    MoveJ pInicioX62_Pinca1, V_rapide, Z_arret, Tool_Pince1\WObj:=wobj_X62;
    !
    ! E13:interferencia2 com K5
    ! O12:fora de interferencia1 com K5
    EVENT\E13;
    ORDRE\O12;
    !
    MoveJ [[602.06,1695.19,2908.36],[0.0694316,-0.00204347,0.00124342,-0.997584],[0,-1,0,0],[59.9379,9E+09,9E+09,9E+09,9E+09,9E+09]], V_rapide, Z_arret, Tool_Pince1\WObj:=wobj_X62;
    !
    ! E13:interferencia2 com K5
    ! O12:fora de interferencia1 com K5
    EVENT\E13;
    ORDRE\O12;
    !
    MoveJ [[1650.02,1566.65,2799.96],[0.370322,0.000249773,0.000216744,-0.928904],[0,0,1,0],[15,9E+09,9E+09,9E+09,9E+09,9E+09]], V_rapide, Z_moyen, Tool_Pince1\WObj:=wobj_X62;
    MoveJ [[2181.41,1327.16,2032.09],[0.381242,0.000299882,0.000125925,-0.924475],[0,0,1,0],[183.538,9E+09,9E+09,9E+09,9E+09,9E+09]], V_rapide, Z_moyen, Tool_Pince1\WObj:=wobj_X62;
    MoveL [[1800.58,758.31,2024.83],[0.381244,0.000300867,0.000120671,-0.924474],[0,0,0,0],[183.538,9E+09,9E+09,9E+09,9E+09,9E+09]], V_rapide, Z_moyen, Tool_Pince1\WObj:=wobj_X62;
    MoveL [[1764.11,614.16,2072.30],[0.381245,0.000303532,0.00010268,-0.924474],[0,0,0,0],[183.538,9E+09,9E+09,9E+09,9E+09,9E+09]], V_rapide, Z_moyen, Tool_Pince1\WObj:=wobj_X62;
    MoveL [[1659.86,663.46,2032.41],[0.381237,0.000301139,0.000117928,-0.924477],[0,0,0,0],[140,9E+09,9E+09,9E+09,9E+09,9E+09]], V_rapide, Z_moyen, Tool_Pince1\WObj:=wobj_X62;
    !
    SR_SOUDER lscs2002942400,V_moyen,1,1,Tool_Pince1,wobj_X62;
    SR_SOUDER lscsg002940402,V_moyen,1,2,Tool_Pince1,wobj_X62;
    SR_SOUDER lscsg002940502,V_moyen,1,2,Tool_Pince1,wobj_X62;
    !
    MoveL [[1888.73,628.89,2158.57],[0.46006,-0.0228879,-0.0118518,-0.887514],[0,-1,0,0],[35.0008,9E+09,9E+09,9E+09,9E+09,9E+09]],V_rapide,Z_moyen,Tool_Pince1\WObj:=wobj_X62;
    MoveL [[2001.09,630.15,2158.77],[0.45992,-0.0313939,-0.0162592,-0.887256],[0,-1,0,0],[35,9E+09,9E+09,9E+09,9E+09,9E+09]],V_rapide,Z_moyen,Tool_Pince1\WObj:=wobj_X62;
    !
    SR_SOUDER lscsg002940602,V_moyen,1,2,Tool_Pince1,wobj_X62;
    SR_SOUDER lscsg002940702,V_moyen,1,2,Tool_Pince1,wobj_X62;
    SR_SOUDER lsdcd002932302, V_moyen, 1, 2, Tool_Pince1, wobj_X62;
    !
    MoveL [[2112.35,622.94,2071.75],[0.601153,0.000260756,1.84552E-05,-0.799134],[0,0,0,0],[134.461,9E+09,9E+09,9E+09,9E+09,9E+09]],V_rapide,Z_moyen,Tool_Pince1\WObj:=wobj_X62;
    MoveL [[2277.78,623.66,2088.68],[0.61438,0.00026062,0.000197661,-0.789011],[0,0,0,0],[99.9998,9E+09,9E+09,9E+09,9E+09,9E+09]],V_rapide,Z_moyen,Tool_Pince1\WObj:=wobj_X62;
    !
    SR_SOUDER lscsg002940802_B,V_moyen,1,2,Tool_Pince1,wobj_X62;
    SR_SOUDER lscsg002940902,V_moyen,1,2,Tool_Pince1,wobj_X62;
    SR_SOUDER lscsg002941002,V_moyen,1,2,Tool_Pince1,wobj_X62;
    !
    MoveL [[2430.75,632.00,2159.24],[0.65197,-0.0151493,-0.013018,-0.757982],[0,-1,0,0],[35,9E+09,9E+09,9E+09,9E+09,9E+09]],V_rapide,Z_moyen,Tool_Pince1\WObj:=wobj_X62;
    MoveL [[2543.78,631.39,2158.47],[0.712277,-0.0103391,-0.0104878,-0.701745],[0,-1,0,0],[34.9994,9E+09,9E+09,9E+09,9E+09,9E+09]],V_rapide,Z_moyen,Tool_Pince1\WObj:=wobj_X62;
    !
    SR_SOUDER lscsg002941202,V_moyen,1,2,Tool_Pince1,wobj_X62;
    !
    MoveL [[2540.85,667.11,2064.42],[0.712277,-0.0103403,-0.0104873,-0.701745],[0,-1,0,0],[168.705,9E+09,9E+09,9E+09,9E+09,9E+09]],V_rapide,Z_moyen,Tool_Pince1\WObj:=wobj_X62;
    MoveL [[2529.75,106.99,2062.78],[0.770678,0.00010718,-5.65434E-05,-0.637225],[0,-1,0,0],[170,9E+09,9E+09,9E+09,9E+09,9E+09]],V_rapide,Z_moyen,Tool_Pince1\WObj:=wobj_X62;
    MoveL [[2798.87,290.44,2173.09],[0.872979,-0.00143955,-0.00186681,-0.487753],[0,-1,-1,0],[44.59,9E+09,9E+09,9E+09,9E+09,9E+09]],V_rapide,Z_arret,Tool_Pince1\WObj:=wobj_X62;
    !
    ! O12:fora de interferencia1 com K5
    ! O13:fora de interferencia2 com K5
    ORDRE\O12\O13;
    !
    MoveL [[2687.98,421.61,2066.53],[0.897783,-0.00356194,-0.00758891,-0.440358],[0,0,-1,0],[170,9E+09,9E+09,9E+09,9E+09,9E+09]],V_rapide,Z_moyen,Tool_Pince1\WObj:=wobj_X62;
    MoveL [[2646.63,666.42,2060.91],[0.921929,-0.00569541,-0.013042,-0.387097],[0,0,-1,0],[160,9E+09,9E+09,9E+09,9E+09,9E+09]],V_rapide,Z_moyen,Tool_Pince1\WObj:=wobj_X62;
    !
    SR_SOUDER lscsg002941302,V_moyen,1,2,Tool_Pince1,wobj_X62;
    !
    MoveL [[2646.63,666.42,2060.91],[0.921929,-0.00569541,-0.013042,-0.387097],[0,0,-1,0],[160,9E+09,9E+09,9E+09,9E+09,9E+09]],V_rapide,Z_moyen,Tool_Pince1\WObj:=wobj_X62;
    MoveL [[2638.67,603.72,2062.9],[0.91586,-9.21472E-05,0.000138523,-0.401498],[0,-1,-1,0],[160,9E+09,9E+09,9E+09,9E+09,9E+09]],V_rapide,Z_moyen,Tool_Pince1\WObj:=wobj_X62;
    MoveL [[2733.77,618.85,2085.50],[0.930262,-0.000109742,0.000151233,-0.366895],[0,-1,-1,0],[160,9E+09,9E+09,9E+09,9E+09,9E+09]], V_rapide, Z_arret, Tool_Pince1\WObj:=wobj_X62;
    !
    ! E12:interferencia1 com K5
    ! O13:fora de interferencia2 com K5
    EVENT\E12;
    ORDRE\O13;
    !
    SR_SOUDER lscs2002948300,V_moyen,1,1,Tool_Pince1,wobj_X62;
    SR_SOUDER lscs2002947600, V_moyen, 1, 1, Tool_Pince1, wobj_X62;
    SR_SOUDER lscs2002948400,V_moyen,1,1,Tool_Pince1,wobj_X62;
    !
    MoveL [[2836.77,664.37,2084.41],[0.930318,-0.000108518,0.000131406,-0.366754],[0,-1,-1,0],[100,9E+09,9E+09,9E+09,9E+09,9E+09]],V_rapide,Z_moyen,Tool_Pince1\WObj:=wobj_X62;
    MoveL [[2847.69,539.48,2094.67],[0.930318,-0.000109137,0.000129915,-0.366755],[0,-1,-1,0],[99.9997,9E+09,9E+09,9E+09,9E+09,9E+09]], V_rapide, Z_moyen, Tool_Pince1\WObj:=wobj_X62;
    !
    SR_SOUDER lscs2002839500_B,V_moyen,1,2,Tool_Pince1,wobj_X62;
    !
    ! E12:interferencia1 com K5
    ! O13:fora de interferencia2 com K5
    EVENT\E12;
    ORDRE\O13;
    !
    MoveL [[2847.68,539.48,2094.66],[0.930318,-0.000107632,0.000130594,-0.366754],[0,-1,-1,0],[99.9985,9E+09,9E+09,9E+09,9E+09,9E+09]],V_rapide,Z_moyen,Tool_Pince1\WObj:=wobj_X62;
    MoveL [[2961.74,544.95,2110.29],[0.920929,0.00770745,-0.00317349,-0.389642],[0,0,-1,0],[99.9985,9E+09,9E+09,9E+09,9E+09,9E+09]], V_rapide, Z_moyen, Tool_Pince1\WObj:=wobj_X62;
    !
    SR_SOUDER lscs2002839600_B,V_moyen,1,2,Tool_Pince1,wobj_X62;
    !
    MoveL [[2961.78,544.91,2096.91],[0.920929,0.00771093,-0.0031708,-0.389642],[0,0,-1,0],[99.9985,9E+09,9E+09,9E+09,9E+09,9E+09]],V_rapide,Z_moyen,Tool_Pince1\WObj:=wobj_X62;
    MoveL [[2953.81,635.94,2096.51],[0.935302,0.00758254,-0.00346754,-0.353752],[0,0,-1,0],[99.9985,9E+09,9E+09,9E+09,9E+09,9E+09]], V_rapide, Z_moyen, Tool_Pince1\WObj:=wobj_X62;
    !
    SR_SOUDER lscs2002947700,V_moyen,1,2,Tool_Pince1,wobj_X62;
    !
    MoveL [[2976.83,612.40,2082.87],[0.93625,-8.88603E-05,0.000120546,-0.351335],[0,-1,-1,0],[160,9E+09,9E+09,9E+09,9E+09,9E+09]],V_rapide,Z_moyen,Tool_Pince1\WObj:=wobj_X62;
    MoveJ [[2868.21,503.75,2082.92],[0.909496,-0.000142875,0.00013103,-0.415712],[0,-1,-1,0],[160,9E+09,9E+09,9E+09,9E+09,9E+09]],V_rapide,Z_moyen,Tool_Pince1\WObj:=wobj_X62;
    MoveL [[2903.89,230.57,2115.02],[0.883552,0.000906724,0.0020198,-0.468328],[0,-1,-1,0],[106.782,9E+09,9E+09,9E+09,9E+09,9E+09]],V_rapide,Z_moyen,Tool_Pince1\WObj:=wobj_X62;
    MoveL [[2725.33,-217.14,2165.65],[0.813387,0.0022139,0.00456468,-0.581701],[0,-1,0,0],[183.878,9E+09,9E+09,9E+09,9E+09,9E+09]],V_rapide,Z_moyen,Tool_Pince1\WObj:=wobj_X62;
    MoveL [[2892.2,-378.24,2080.12],[0.820879,0.00325637,0.00569146,-0.571065],[0,-1,0,0],[170,9E+09,9E+09,9E+09,9E+09,9E+09]],V_rapide,Z_moyen,Tool_Pince1\WObj:=wobj_X62;
    MoveL [[3180.5,-656.48,2080],[0.833499,0.00504519,0.00760941,-0.552446],[0,0,0,0],[170,9E+09,9E+09,9E+09,9E+09,9E+09]],V_rapide,Z_moyen,Tool_Pince1\WObj:=wobj_X62;
    !
    SR_SOUDER lscsg002952001, V_moyen, 1, 3, Tool_Pince1, wobj_X62;
    SR_SOUDER lscs1002947400,V_moyen,1,2,Tool_Pince1,wobj_X62;
    SR_SOUDER lscs1002947300,V_moyen,1,2,Tool_Pince1,wobj_X62;
    !
    MoveL [[2959.66,-658.22,2080],[0.826002,1.26628E-06,-6.1516E-09,-0.563667],[0,-1,-1,0],[160,9E+09,9E+09,9E+09,9E+09,9E+09]],V_rapide,Z_moyen,Tool_Pince1\WObj:=wobj_X62;
    MoveL [[2957.72,-527.54,2087.24],[0.856587,0.0240609,0.014427,-0.51524],[0,0,-1,0],[160,9E+09,9E+09,9E+09,9E+09,9E+09]],V_rapide,Z_moyen,Tool_Pince1\WObj:=wobj_X62;
    !
    SR_SOUDER lscs1002839400_B,V_moyen,1,2,Tool_Pince1,wobj_X62;
    SR_SOUDER lspac002893200,V_moyen,1,1,Tool_Pince1,wobj_X62;
    SR_SOUDER lspac002893300,V_moyen,1,1,Tool_Pince1,wobj_X62;
    SR_SOUDER lspac002893400,V_moyen,1,1,Tool_Pince1,wobj_X62;
    SR_SOUDER lspac006169000,V_moyen,1,1,Tool_Pince1,wobj_X62;
    SR_SOUDER lspac002893500,V_moyen,1,1,Tool_Pince1,wobj_X62;
    SR_SOUDER lspac006167800,V_moyen,1,1,Tool_Pince1,wobj_X62;
    SR_SOUDER lspac002893600,V_moyen,1,1,Tool_Pince1,wobj_X62;
    SR_SOUDER lspac002893700,V_moyen,1,1,Tool_Pince1,wobj_X62;
    SR_SOUDER lspac002893800,V_moyen,1,1,Tool_Pince1,wobj_X62;
    !
    MoveL [[2958.19,527.03,2127.56],[0.919306,-0.0378263,-0.0331513,-0.390315],[0,-1,-1,0],[160,9E+09,9E+09,9E+09,9E+09,9E+09]], V_moyen, Z_moyen, Tool_Pince1\WObj:=wobj_X62;
    MoveL [[2862.51,513.76,2127.39],[0.9045,-0.0491103,-0.0197838,-0.423175],[0,-1,-1,0],[160,9E+09,9E+09,9E+09,9E+09,9E+09]], V_moyen, Z_moyen, Tool_Pince1\WObj:=wobj_X62;
    !
    SR_SOUDER lspac002893100,V_moyen,1,1,Tool_Pince1,wobj_X62;
    !
    MoveL [[2857.80,455.64,2170.88],[0.904867,-0.0141977,0.000985929,-0.425456],[0,-1,-1,0],[37.3852,9E+09,9E+09,9E+09,9E+09,9E+09]],V_rapide,Z_moyen,Tool_Pince1\WObj:=wobj_X62;
    !
    SR_SOUDER lspac002893000,V_moyen,1,1,Tool_Pince1,wobj_X62;
    SR_SOUDER lspac002892900,V_moyen,1,1,Tool_Pince1,wobj_X62;
    SR_SOUDER lspac006168400,V_moyen,1,1,Tool_Pince1,wobj_X62;
    SR_SOUDER lspac002892800,V_moyen,1,1,Tool_Pince1,wobj_X62;
    SR_SOUDER lspac006169600,V_moyen,1,1,Tool_Pince1,wobj_X62;
    SR_SOUDER lspac002892700,V_moyen,1,1,Tool_Pince1,wobj_X62;
    SR_SOUDER lspac002892600,V_moyen,1,1,Tool_Pince1,wobj_X62;
    SR_SOUDER lspac002892500,V_moyen,1,1,Tool_Pince1,wobj_X62;
    SR_SOUDER lscs1002839300_B,V_moyen,1,2,Tool_Pince1,wobj_X62;
    !
    MoveL [[2858.38,-489.28,2086.28],[0.832504,0.0281077,0.0314063,-0.552414],[0,0,-1,0],[170,9E+09,9E+09,9E+09,9E+09,9E+09]],V_rapide,Z_moyen,Tool_Pince1\WObj:=wobj_X62;
    MoveL [[2836.28,-656.22,2069.50],[0.815223,5.65403E-06,7.3518E-06,-0.579147],[0,-1,0,0],[160,9E+09,9E+09,9E+09,9E+09,9E+09]],V_rapide,Z_moyen,Tool_Pince1\WObj:=wobj_X62;
    !
    SR_SOUDER lsdc1002933000, V_moyen, 1, 2, Tool_Pince1, wobj_X62;
    SR_SOUDER lscs1002947200,V_moyen,1,2,Tool_Pince1,wobj_X62;
    SR_SOUDER lscs1002947100,V_moyen,1,2,Tool_Pince1,wobj_X62;
    !
    MoveL [[2737.02,-598.43,2063.08],[0.804154,1.14616E-05,2.43119E-06,-0.594422],[0,-1,0,0],[160,9E+09,9E+09,9E+09,9E+09,9E+09]],V_rapide,Z_moyen,Tool_Pince1\WObj:=wobj_X62;
    MoveL [[2638.91,-600.76,2063.08],[0.804155,1.61702E-06,2.0742E-06,-0.59442],[0,-1,-1,0],[160,9E+09,9E+09,9E+09,9E+09,9E+09]],V_rapide,Z_moyen,Tool_Pince1\WObj:=wobj_X62;
    !
    SR_SOUDER lscs1002942300,V_moyen,1,1,Tool_Pince1,wobj_X62;
    SR_SOUDER lscsd002941201,V_moyen,1,2,Tool_Pince1,wobj_X62;
    !
    ! O12:fora de interferencia1 com K5
    ! O13:fora de interferencia2 com K5
    ORDRE\O12\O13;
    !
    SR_SOUDER lscsd002941001,V_moyen,1,2,Tool_Pince1,wobj_X62;
    SR_SOUDER lscsd002940901,V_moyen,1,2,Tool_Pince1,wobj_X62;
    SR_SOUDER lscsd002940801,V_moyen,1,2,Tool_Pince1,wobj_X62;
    SR_SOUDER lsdcg002932401, V_moyen, 1, 2, Tool_Pince1, wobj_X62;
    !
    MoveL [[2250.91,-658.34,2071.74],[0.713315,-7.82072E-07,-3.16574E-06,-0.700844],[0,-1,0,0],[160,9E+09,9E+09,9E+09,9E+09,9E+09]],V_rapide,Z_moyen,Tool_Pince1\WObj:=wobj_X62;
    MoveL [[2235.49,-509.78,2082.81],[0.695343,0.0282441,0.0285761,-0.717555],[0,0,0,0],[160,9E+09,9E+09,9E+09,9E+09,9E+09]],V_rapide,Z_moyen,Tool_Pince1\WObj:=wobj_X62;
    !
    SR_SOUDER lscs1002839000_B,V_moyen,1,2,Tool_Pince1,wobj_X62;
    SR_SOUDER lspac002890400,V_moyen,1,1,Tool_Pince1,wobj_X62;
    SR_SOUDER lspac002890500,V_moyen,1,1,Tool_Pince1,wobj_X62;
    SR_SOUDER lspac002890600,V_moyen,1,1,Tool_Pince1,wobj_X62;
    SR_SOUDER lspac006168800,V_moyen,1,1,Tool_Pince1,wobj_X62;
    SR_SOUDER lspac002890700,V_moyen,1,1,Tool_Pince1,wobj_X62;
    SR_SOUDER lspac006167600,V_moyen,1,1,Tool_Pince1,wobj_X62;
    SR_SOUDER lspac002890800,V_moyen,1,1,Tool_Pince1,wobj_X62;
    SR_SOUDER lspac002890900,V_moyen,1,1,Tool_Pince1,wobj_X62;
    SR_SOUDER lspac002891000,V_moyen,1,1,Tool_Pince1,wobj_X62;
    SR_SOUDER lscs2002839200_B,V_moyen,1,2,Tool_Pince1,wobj_X62;
    !
    MoveL [[2235.13,533.73,2100],[0.695057,-0.0343774,-0.0362408,-0.717217],[0,-1,0,0],[160,9E+09,9E+09,9E+09,9E+09,9E+09]],V_rapide,Z_moyen,Tool_Pince1\WObj:=wobj_X62;
    MoveL [[2126.59,525.70,2089.46],[0.658646,-0.0167254,-0.0210119,-0.751974],[0,-1,0,0],[160,9E+09,9E+09,9E+09,9E+09,9E+09]], V_rapide, Z_moyen, Tool_Pince1\WObj:=wobj_X62;
    !
    SR_SOUDER lscs2002839100_B,V_moyen,1,2,Tool_Pince1,wobj_X62;
    SR_SOUDER lspac002890300,V_moyen,1,1,Tool_Pince1,wobj_X62;
    SR_SOUDER lspac002890200,V_moyen,1,1,Tool_Pince1,wobj_X62;
    SR_SOUDER lspac002890100,V_moyen,1,1,Tool_Pince1,wobj_X62;
    SR_SOUDER lspac006168200,V_moyen,1,1,Tool_Pince1,wobj_X62;
    SR_SOUDER lspac002890000,V_moyen,1,1,Tool_Pince1,wobj_X62;
    SR_SOUDER lspac006169400,V_moyen,1,1,Tool_Pince1,wobj_X62;
    SR_SOUDER lspac002889900,V_moyen,1,1,Tool_Pince1,wobj_X62;
    SR_SOUDER lspac002889800,V_moyen,1,1,Tool_Pince1,wobj_X62;
    SR_SOUDER lspac002889700,V_moyen,1,1,Tool_Pince1,wobj_X62;
    SR_SOUDER lscs1002838900_B,V_moyen,1,2,Tool_Pince1,wobj_X62;
    !
    MoveL [[2135.27,-514.17,2084.58],[0.707903,0.0308484,0.0366874,-0.704681],[0,0,0,0],[160,9E+09,9E+09,9E+09,9E+09,9E+09]],V_rapide,Z_moyen,Tool_Pince1\WObj:=wobj_X62;
    MoveL [[2145.10,-626.48,2085.09],[0.707903,0.030849,0.036688,-0.704682],[0,0,0,0],[160,9E+09,9E+09,9E+09,9E+09,9E+09]],V_rapide,Z_moyen,Tool_Pince1\WObj:=wobj_X62;
    !
    SR_SOUDER lsdcg002932301, V_moyen, 1, 2, Tool_Pince1, wobj_X62;
    SR_SOUDER lscsd002940701,V_moyen,1,2,Tool_Pince1,wobj_X62;
    SR_SOUDER lscsd002940601,V_moyen,1,2,Tool_Pince1,wobj_X62;
    SR_SOUDER lscsd002940501,V_moyen,1,2,Tool_Pince1,wobj_X62;
    SR_SOUDER lscsd002940401,V_moyen,1,2,Tool_Pince1,wobj_X62;
    !
    MoveL [[1769.05,-537.66,2062.91],[0.62095,-1.33124E-06,-4.31943E-06,-0.78385],[0,-1,0,0],[170,9E+09,9E+09,9E+09,9E+09,9E+09]],V_rapide,Z_moyen,Tool_Pince1\WObj:=wobj_X62;
    MoveL [[1470.09,-502.91,2081.97],[0.520364,0.0154325,0.0248961,-0.853442],[0,0,0,0],[160,9E+09,9E+09,9E+09,9E+09,9E+09]],V_rapide,Z_moyen,Tool_Pince1\WObj:=wobj_X62;
    MoveL [[1432.88,-492.27,2156.85],[0.520088,0.0239709,0.0300975,-0.853245],[0,0,0,0],[66.9765,9E+09,9E+09,9E+09,9E+09,9E+09]],V_rapide,Z_moyen,Tool_Pince1\WObj:=wobj_X62;
    !
    SR_SOUDER lscs1002838200_B,V_moyen,1,2,Tool_Pince1,wobj_X62;
    SR_SOUDER lspac002867100,V_moyen,1,1,Tool_Pince1,wobj_X62;
    SR_SOUDER lspac002867200,V_moyen,1,1,Tool_Pince1,wobj_X62;
    SR_SOUDER lspac006171300_B,V_moyen,1,1,Tool_Pince1,wobj_X62;
    !
    MoveL [[1427.18,-389.85,2089.13],[0.520563,0.00960129,0.015755,-0.853624],[0,0,0,0],[160,9E+09,9E+09,9E+09,9E+09,9E+09]],V_rapide,Z_moyen,Tool_Pince1\WObj:=wobj_X62;
    MoveL [[1453.86,-198.92,2110.29],[0.520654,0.00529497,0.00880381,-0.853706],[0,0,0,0],[183.227,9E+09,9E+09,9E+09,9E+09,9E+09]],V_rapide,Z_moyen,Tool_Pince1\WObj:=wobj_X62;
    !
    SR_SOUDER lspac002867300,V_moyen,1,1,Tool_Pince1,wobj_X62;
    SR_SOUDER lspac004679300,V_moyen,1,1,Tool_Pince1,wobj_X62;
    SR_SOUDER lspac006171700,V_moyen,1,1,Tool_Pince1,wobj_X62;
    SR_SOUDER lspac002867400,V_moyen,1,1,Tool_Pince1,wobj_X62;
    SR_SOUDER lspac002867500,V_moyen,1,1,Tool_Pince1,wobj_X62;
    !
    MoveL [[1427.46,199.95,2087.77],[0.460873,-0.00466668,-0.0086408,-0.887412],[0,-1,0,0],[160,9E+09,9E+09,9E+09,9E+09,9E+09]],V_rapide,Z_moyen,Tool_Pince1\WObj:=wobj_X62;
    MoveL [[1429.24,375.03,2090.92],[0.437051,-0.0019001,-0.0438692,-0.898364],[0,0,0,0],[182.475,9E+09,9E+09,9E+09,9E+09,9E+09]], V_moyen, Z_petit, Tool_Pince1\WObj:=wobj_X62;
    !
    SR_SOUDER lspac006172100_B,V_moyen,1,1,Tool_Pince1,wobj_X62;
    SR_SOUDER lspac002867600,V_moyen,1,1,Tool_Pince1,wobj_X62;
    SR_SOUDER lspac002867700,V_moyen,1,1,Tool_Pince1,wobj_X62;
    SR_SOUDER lscs2002838400_B,V_moyen,1,2,Tool_Pince1,wobj_X62;
    !
    MoveL [[1432.15,527.47,2071.51],[0.353061,-0.0165696,-0.0612235,-0.933448],[0,-1,0,0],[160,9E+09,9E+09,9E+09,9E+09,9E+09]], V_rapide, Z_moyen, Tool_Pince1\WObj:=wobj_X62;
    MoveL [[1320.78,516.51,2071.30],[0.318701,-0.0159195,-0.0302608,-0.947239],[0,-1,0,0],[160,9E+09,9E+09,9E+09,9E+09,9E+09]],V_rapide,Z_moyen,Tool_Pince1\WObj:=wobj_X62;
    !
    SR_SOUDER lscs2002838300,V_moyen,1,2,Tool_Pince1,wobj_X62;
    SR_SOUDER lspac002872000,V_moyen,1,2,Tool_Pince1,wobj_X62;
    SR_SOUDER lspac002871900,V_moyen,1,1,Tool_Pince1,wobj_X62;
    SR_SOUDER lspac002871800,V_moyen,1,2,Tool_Pince1,wobj_X62;
    SR_SOUDER lspac002871700,V_moyen,1,2,Tool_Pince1,wobj_X62;
    SR_SOUDER lspac002871600,V_moyen,1,2,Tool_Pince1,wobj_X62;
    SR_SOUDER lspac002871500,V_moyen,1,2,Tool_Pince1,wobj_X62;
    SR_SOUDER lspac002871400,V_moyen,1,2,Tool_Pince1,wobj_X62;
    SR_SOUDER lspac002871300,V_moyen,1,1,Tool_Pince1,wobj_X62;
    SR_SOUDER lspac002871200,V_moyen,1,2,Tool_Pince1,wobj_X62;
    SR_SOUDER lspac002871100,V_moyen,1,2,Tool_Pince1,wobj_X62;
    SR_SOUDER lspac002871000,V_moyen,1,2,Tool_Pince1,wobj_X62;
    SR_SOUDER lspac002870900,V_moyen,1,2,Tool_Pince1,wobj_X62;
    ! Abrir Grampos
    !
  ENDPROC

  PROC T_X62K3E23H2()
    VAR bool bStatus;
    Aff_Traj "T_X62K3E23H2";
    AntiReboucle;

    MoveJ pInicioX62_Pinca1, V_rapide, Z_arret, Tool_Pince1\WObj:=wobj_X62;
    !
    ! E13:interferencia2 com K5
    ! O12:fora de interferencia1 com K5
    EVENT\E13;
    ORDRE\O12;
    !
    MoveJ [[602.06,1695.19,2908.36],[0.0694316,-0.00204347,0.00124342,-0.997584],[0,-1,0,0],[59.9379,9E+09,9E+09,9E+09,9E+09,9E+09]], V_rapide, Z_arret, Tool_Pince1\WObj:=wobj_X62;
    !
    ! E13:interferencia2 com K5
    ! O12:fora de interferencia1 com K5
    EVENT\E13;
    ORDRE\O12;
    !
    MoveJ [[1650.02,1566.65,2799.96],[0.370322,0.000249773,0.000216744,-0.928904],[0,0,1,0],[15,9E+09,9E+09,9E+09,9E+09,9E+09]], V_rapide, Z_moyen, Tool_Pince1\WObj:=wobj_X62;
    MoveJ [[2181.41,1327.16,2032.09],[0.381242,0.000299882,0.000125925,-0.924475],[0,0,1,0],[183.538,9E+09,9E+09,9E+09,9E+09,9E+09]], V_rapide, Z_moyen, Tool_Pince1\WObj:=wobj_X62;
    MoveL [[2140.22,1267.39,1974.98],[0.380608,0.000250388,0.000124268,-0.924737],[0,0,1,0],[183.342,9E+09,9E+09,9E+09,9E+09,9E+09]], V_rapide, Z_moyen, Tool_Pince1\WObj:=wobj_X62;
    MoveL [[1764.22,613.94,2018.73],[0.381236,0.000302116,0.000105547,-0.924478],[0,0,0,0],[183.537,9E+09,9E+09,9E+09,9E+09,9E+09]], V_rapide, Z_moyen, Tool_Pince1\WObj:=wobj_X62;
    MoveL [[1659.86,663.46,2032.41],[0.381237,0.000301139,0.000117928,-0.924477],[0,0,0,0],[140,9E+09,9E+09,9E+09,9E+09,9E+09]], V_rapide, Z_moyen, Tool_Pince1\WObj:=wobj_X62;
    !
    SR_SOUDER lscs2002942400, V_moyen, 1, 15, Tool_Pince1, wobj_X62;
    SR_SOUDER lscsg002940402, V_moyen, 1, 15, Tool_Pince1, wobj_X62;
    SR_SOUDER lscsg002940502, V_moyen, 1, 15, Tool_Pince1, wobj_X62;
    !
    MoveL [[1889.96,614.75,2158.61],[0.46006,-0.0228897,-0.0118453,-0.887514],[0,-1,0,0],[35.001,9E+09,9E+09,9E+09,9E+09,9E+09]],V_rapide,Z_moyen,Tool_Pince1\WObj:=wobj_X62;
    MoveL [[2002.32,616.22,2158.84],[0.45992,-0.0313938,-0.0162634,-0.887256],[0,-1,0,0],[35,9E+09,9E+09,9E+09,9E+09,9E+09]],V_rapide,Z_moyen,Tool_Pince1\WObj:=wobj_X62;
    !
    SR_SOUDER lscsg002940602, V_moyen, 1, 15, Tool_Pince1, wobj_X62;
    SR_SOUDER lscsg002940702, V_moyen, 1, 15, Tool_Pince1, wobj_X62;
    SR_SOUDER lsdcd002932302, V_moyen, 1, 15, Tool_Pince1, wobj_X62;
    !
    MoveL [[2112.35,622.94,2071.75],[0.601153,0.000260756,1.84552E-05,-0.799134],[0,0,0,0],[134.461,9E+09,9E+09,9E+09,9E+09,9E+09]],V_rapide,Z_moyen,Tool_Pince1\WObj:=wobj_X62;
    MoveL [[2247.75,623.68,2092.80],[0.614378,0.000259002,0.000201606,-0.789012],[0,0,0,0],[99.9998,9E+09,9E+09,9E+09,9E+09,9E+09]],V_rapide,Z_moyen,Tool_Pince1\WObj:=wobj_X62;
    !
    SR_SOUDER lscsg002940802, V_moyen, 1, 15, Tool_Pince1, wobj_X62;
    SR_SOUDER lscsg002940902, V_moyen, 1, 15, Tool_Pince1, wobj_X62;
    SR_SOUDER lscsg002941002, V_moyen, 1, 15, Tool_Pince1, wobj_X62;
    SR_SOUDER lscsg002941202, V_moyen, 1, 15, Tool_Pince1, wobj_X62;
    !
    MoveL [[2529.75,106.98,2162.76],[0.74488,0.000109833,-5.00299E-05,-0.667199],[0,0,0,0],[61.2346,9E+09,9E+09,9E+09,9E+09,9E+09]],V_rapide,Z_moyen,Tool_Pince1\WObj:=wobj_X62;
    MoveL [[2798.87,290.44,2173.09],[0.872979,-0.00143955,-0.00186681,-0.487753],[0,-1,-1,0],[44.59,9E+09,9E+09,9E+09,9E+09,9E+09]],V_rapide,Z_arret,Tool_Pince1\WObj:=wobj_X62;
    !
    ! O12:fora de interferencia1 com K5
    ! O13:fora de interferencia2 com K5
    ORDRE\O12\O13;
    !
    MoveL [[2687.99,421.61,2164.62],[0.897784,-0.00356148,-0.0075883,-0.440357],[0,0,-1,0],[39.7045,9E+09,9E+09,9E+09,9E+09,9E+09]],V_rapide,Z_moyen,Tool_Pince1\WObj:=wobj_X62;
    !
    SR_SOUDER lscsg002941302, V_moyen, 1, 15, Tool_Pince1, wobj_X62;
    !
    MoveL [[2638.67,603.72,2162.90],[0.91586,-9.21472E-05,0.000138523,-0.401498],[0,-1,-1,0],[39.9998,9E+09,9E+09,9E+09,9E+09,9E+09]],V_rapide,Z_moyen,Tool_Pince1\WObj:=wobj_X62;
    MoveL [[2736.74,585.39,2162.84],[0.930263,-9.92501E-05,0.000159226,-0.366894],[0,-1,-1,0],[40.0001,9E+09,9E+09,9E+09,9E+09,9E+09]], V_rapide, Z_arret, Tool_Pince1\WObj:=wobj_X62;
    !
    ! E12:interferencia1 com K5
    ! O13:fora de interferencia2 com K5
    EVENT\E12;
    ORDRE\O13;
    !
    SR_SOUDER lscs2002948300,V_moyen,1,1,Tool_Pince1,wobj_X62;
    SR_SOUDER lscs2002947600, V_moyen, 1, 1, Tool_Pince1, wobj_X62;
    SR_SOUDER lscs2002948400,V_moyen,1,1,Tool_Pince1,wobj_X62;
    !
    ! E12:interferencia1 com K5
    ! O13:fora de interferencia2 com K5
    EVENT\E12;
    ORDRE\O13;
    !
    MoveL [[2836.77,664.36,2084.43],[0.930318,-0.000111582,0.00012884,-0.366755],[0,-1,-1,0],[99.9999,9E+09,9E+09,9E+09,9E+09,9E+09]],V_rapide,Z_moyen,Tool_Pince1\WObj:=wobj_X62;
    MoveL [[2978.75,664.36,2072.80],[0.956803,-0.000109625,0.000180293,-0.290739],[0,-1,-1,0],[99.9999,9E+09,9E+09,9E+09,9E+09,9E+09]],V_rapide,Z_moyen,Tool_Pince1\WObj:=wobj_X62;
    !
    SR_SOUDER lscs2002947700,V_moyen,1,2,Tool_Pince1,wobj_X62;
    SR_SOUDER lscs2002947700_1, V_moyen, 1, 2, Tool_Pince1, wobj_X62;
    !
    MoveL [[2976.82,612.40,2162.87],[0.930798,-9.10824E-05,0.000119097,-0.365534],[0,-1,-1,0],[40.0001,9E+09,9E+09,9E+09,9E+09,9E+09]],V_rapide,Z_moyen,Tool_Pince1\WObj:=wobj_X62;
    MoveL [[3032.03,552.56,2164.42],[0.924331,-7.91105E-05,0.000121254,-0.381592],[0,-1,-1,0],[39.8012,9E+09,9E+09,9E+09,9E+09,9E+09]],V_rapide,Z_moyen,Tool_Pince1\WObj:=wobj_X62;
    MoveL [[2903.89,230.57,2115.02],[0.883552,0.000906724,0.0020198,-0.468328],[0,-1,-1,0],[106.782,9E+09,9E+09,9E+09,9E+09,9E+09]],V_rapide,Z_moyen,Tool_Pince1\WObj:=wobj_X62;
    MoveL [[2725.33,-217.14,2165.65],[0.813387,0.0022139,0.00456468,-0.581701],[0,-1,0,0],[183.878,9E+09,9E+09,9E+09,9E+09,9E+09]],V_rapide,Z_moyen,Tool_Pince1\WObj:=wobj_X62;
    MoveL [[2892.20,-378.24,2145.12],[0.820879,0.00325637,0.00569146,-0.571065],[0,-1,0,0],[129.315,9E+09,9E+09,9E+09,9E+09,9E+09]],V_rapide,Z_moyen,Tool_Pince1\WObj:=wobj_X62;
    !
    SR_SOUDER lscsg002952001, V_moyen, 1, 15, Tool_Pince1, wobj_X62;
    SR_SOUDER lscs1002947400, V_moyen, 1, 15, Tool_Pince1, wobj_X62;
    SR_SOUDER lscs1002947400_1, V_moyen, 1, 15, Tool_Pince1, wobj_X62;
    SR_SOUDER lscs1002947300, V_moyen, 1, 15, Tool_Pince1, wobj_X62;
    SR_SOUDER lscs1002839400,V_moyen,1,2,Tool_Pince1,wobj_X62;
    SR_SOUDER lspac002893200,V_moyen,1,1,Tool_Pince1,wobj_X62;
    SR_SOUDER lspac002893300,V_moyen,1,1,Tool_Pince1,wobj_X62;
    SR_SOUDER lspac002893400,V_moyen,1,1,Tool_Pince1,wobj_X62;
    SR_SOUDER lspac006169000,V_moyen,1,1,Tool_Pince1,wobj_X62;
    SR_SOUDER lspac002893500,V_moyen,1,1,Tool_Pince1,wobj_X62;
    SR_SOUDER lspac006167800,V_moyen,1,1,Tool_Pince1,wobj_X62;
    SR_SOUDER lspac002893600,V_moyen,1,1,Tool_Pince1,wobj_X62;
    SR_SOUDER lspac002893700,V_moyen,1,1,Tool_Pince1,wobj_X62;
    SR_SOUDER lspac002893800,V_moyen,1,1,Tool_Pince1,wobj_X62;
    SR_SOUDER lscs2002839600,V_moyen,1,2,Tool_Pince1,wobj_X62;
    !
    MoveL [[2956.89,578.06,2102.81],[0.934244,-0.0245846,-0.00556889,-0.355743],[0,-1,-1,0],[100,9E+09,9E+09,9E+09,9E+09,9E+09]],V_rapide,Z_moyen,Tool_Pince1\WObj:=wobj_X62;
    MoveL [[2857.12,578.03,2098.68],[0.934191,-0.0247615,-0.00622529,-0.35586],[0,-1,-1,0],[99.9999,9E+09,9E+09,9E+09,9E+09,9E+09]],V_rapide,Z_moyen,Tool_Pince1\WObj:=wobj_X62;
    !
    SR_SOUDER lscs2002839500,V_moyen,1,2,Tool_Pince1,wobj_X62;
    SR_SOUDER lspac002893100,V_moyen,1,1,Tool_Pince1,wobj_X62;
    !
    MoveL [[2857.80,455.64,2170.88],[0.904867,-0.0141977,0.000985929,-0.425456],[0,-1,-1,0],[37.3852,9E+09,9E+09,9E+09,9E+09,9E+09]],V_rapide,Z_moyen,Tool_Pince1\WObj:=wobj_X62;
    !
    SR_SOUDER lspac002893000,V_moyen,1,1,Tool_Pince1,wobj_X62;
    SR_SOUDER lspac002892900,V_moyen,1,1,Tool_Pince1,wobj_X62;
    SR_SOUDER lspac006168400,V_moyen,1,1,Tool_Pince1,wobj_X62;
    SR_SOUDER lspac002892800,V_moyen,1,1,Tool_Pince1,wobj_X62;
    SR_SOUDER lspac006169600,V_moyen,1,1,Tool_Pince1,wobj_X62;
    SR_SOUDER lspac002892700,V_moyen,1,1,Tool_Pince1,wobj_X62;
    SR_SOUDER lspac002892600,V_moyen,1,1,Tool_Pince1,wobj_X62;
    SR_SOUDER lspac002892500,V_moyen,1,1,Tool_Pince1,wobj_X62;
    SR_SOUDER lscs1002839300,V_moyen,1,2,Tool_Pince1,wobj_X62;
    !
    MoveL [[2859.00,-619.86,2161.00],[0.820982,0.0101897,0.00686966,-0.570822],[0,0,-1,0],[60.0001,9E+09,9E+09,9E+09,9E+09,9E+09]],V_rapide,Z_moyen,Tool_Pince1\WObj:=wobj_X62;
    !
    SR_SOUDER lsdc1002933000, V_moyen, 1, 15, Tool_Pince1, wobj_X62;
    SR_SOUDER lscs1002947200, V_moyen, 1, 15, Tool_Pince1, wobj_X62;
    SR_SOUDER lscs1002947100, V_moyen, 1, 15, Tool_Pince1, wobj_X62;
    !
    MoveL [[2737.02,-598.43,2163.08],[0.804154,1.14616E-05,2.43119E-06,-0.594422],[0,-1,0,0],[40.0001,9E+09,9E+09,9E+09,9E+09,9E+09]],V_rapide,Z_moyen,Tool_Pince1\WObj:=wobj_X62;
    MoveL [[2638.91,-600.76,2163.08],[0.804155,1.61702E-06,2.0742E-06,-0.59442],[0,-1,-1,0],[39.9998,9E+09,9E+09,9E+09,9E+09,9E+09]],V_rapide,Z_moyen,Tool_Pince1\WObj:=wobj_X62;
    !
    SR_SOUDER lscs1002942300, V_moyen, 1, 15, Tool_Pince1, wobj_X62;
    SR_SOUDER lscsd002941201, V_moyen, 1, 15, Tool_Pince1, wobj_X62;
    !
    ! O12:fora de interferencia1 com K5
    ! O13:fora de interferencia2 com K5
    ORDRE\O12\O13;
    !
    SR_SOUDER lscsd002941001, V_moyen, 1, 15, Tool_Pince1, wobj_X62;
    SR_SOUDER lscsd002940901, V_moyen, 1, 15, Tool_Pince1, wobj_X62;
    SR_SOUDER lscsd002940801, V_moyen, 1, 15, Tool_Pince1, wobj_X62;
    SR_SOUDER lsdcg002932401, V_moyen, 1, 15, Tool_Pince1, wobj_X62;
    SR_SOUDER lscs1002839000,V_moyen,1,2,Tool_Pince1,wobj_X62;
    SR_SOUDER lspac002890400,V_moyen,1,1,Tool_Pince1,wobj_X62;
    SR_SOUDER lspac002890500,V_moyen,1,1,Tool_Pince1,wobj_X62;
    SR_SOUDER lspac002890600,V_moyen,1,1,Tool_Pince1,wobj_X62;
    SR_SOUDER lspac006168800,V_moyen,1,1,Tool_Pince1,wobj_X62;
    SR_SOUDER lspac002890700,V_moyen,1,1,Tool_Pince1,wobj_X62;
    SR_SOUDER lspac006167600,V_moyen,1,1,Tool_Pince1,wobj_X62;
    SR_SOUDER lspac002890800,V_moyen,1,1,Tool_Pince1,wobj_X62;
    SR_SOUDER lspac002890900,V_moyen,1,1,Tool_Pince1,wobj_X62;
    SR_SOUDER lspac002891000,V_moyen,1,1,Tool_Pince1,wobj_X62;
    SR_SOUDER lscs2002839200,V_moyen,1,2,Tool_Pince1,wobj_X62;
    !
    MoveL [[2229.91,578.30,2100.11],[0.613972,-0.01796,-0.0231624,-0.788784],[0,-1,0,0],[101.503,9E+09,9E+09,9E+09,9E+09,9E+09]],V_rapide,Z_moyen,Tool_Pince1\WObj:=wobj_X62;
    MoveL [[2130.14,578.42,2100.87],[0.601034,-0.0175801,-0.0234612,-0.798686],[0,-1,0,0],[101.608,9E+09,9E+09,9E+09,9E+09,9E+09]],V_rapide,Z_moyen,Tool_Pince1\WObj:=wobj_X62;
    !
    SR_SOUDER lscs2002839100,V_moyen,1,2,Tool_Pince1,wobj_X62;
    SR_SOUDER lspac002890300,V_moyen,1,1,Tool_Pince1,wobj_X62;
    SR_SOUDER lspac002890200,V_moyen,1,1,Tool_Pince1,wobj_X62;
    SR_SOUDER lspac002890100,V_moyen,1,1,Tool_Pince1,wobj_X62;
    SR_SOUDER lspac006168200,V_moyen,1,1,Tool_Pince1,wobj_X62;
    SR_SOUDER lspac002890000,V_moyen,1,1,Tool_Pince1,wobj_X62;
    SR_SOUDER lspac006169400,V_moyen,1,1,Tool_Pince1,wobj_X62;
    SR_SOUDER lspac002889900,V_moyen,1,1,Tool_Pince1,wobj_X62;
    SR_SOUDER lspac002889800,V_moyen,1,1,Tool_Pince1,wobj_X62;
    SR_SOUDER lspac002889700,V_moyen,1,1,Tool_Pince1,wobj_X62;
    SR_SOUDER lscs1002838900,V_moyen,1,2,Tool_Pince1,wobj_X62;
    SR_SOUDER lsdcg002932301, V_moyen, 1, 15, Tool_Pince1, wobj_X62;
    SR_SOUDER lscsd002940701, V_moyen, 1, 15, Tool_Pince1, wobj_X62;
    SR_SOUDER lscsd002940601, V_moyen, 1, 15, Tool_Pince1, wobj_X62;
    SR_SOUDER lscsd002940501, V_moyen, 1, 15, Tool_Pince1, wobj_X62;
    SR_SOUDER lscsd002940401, V_moyen, 1, 15, Tool_Pince1, wobj_X62;
    !
    MoveL [[1767.34,-518.18,2162.78],[0.62095,2.70524E-06,5.015E-06,-0.78385],[0,-1,0,0],[40.0003,9E+09,9E+09,9E+09,9E+09,9E+09]],V_rapide,Z_moyen,Tool_Pince1\WObj:=wobj_X62;
    MoveL [[1469.63,-497.72,2181.94],[0.520364,0.0154309,0.0248939,-0.853442],[0,0,0,0],[40.0001,9E+09,9E+09,9E+09,9E+09,9E+09]],V_rapide,Z_moyen,Tool_Pince1\WObj:=wobj_X62;
    !
    SR_SOUDER lscs1002838200,V_moyen,1,2,Tool_Pince1,wobj_X62;
    SR_SOUDER lspac002867100,V_moyen,1,1,Tool_Pince1,wobj_X62;
    SR_SOUDER lspac002867200,V_moyen,1,1,Tool_Pince1,wobj_X62;
    SR_SOUDER lspac006171300,V_moyen,1,1,Tool_Pince1,wobj_X62;
    SR_SOUDER lspac002867300,V_moyen,1,1,Tool_Pince1,wobj_X62;
    SR_SOUDER lspac004679300,V_moyen,1,1,Tool_Pince1,wobj_X62;
    SR_SOUDER lspac006171700,V_moyen,1,1,Tool_Pince1,wobj_X62;
    SR_SOUDER lspac002867400,V_moyen,1,1,Tool_Pince1,wobj_X62;
    SR_SOUDER lspac002867500,V_moyen,1,1,Tool_Pince1,wobj_X62;
    SR_SOUDER lspac006172100,V_moyen,1,1,Tool_Pince1,wobj_X62;
    SR_SOUDER lspac002867600,V_moyen,1,1,Tool_Pince1,wobj_X62;
    SR_SOUDER lspac002867700,V_moyen,1,1,Tool_Pince1,wobj_X62;
    SR_SOUDER lscs2002838400,V_moyen,1,2,Tool_Pince1,wobj_X62;
    !
    MoveL [[1425.97,577.72,2083.22],[0.340978,-0.00978989,-0.0275822,-0.939616],[0,-1,0,0],[127.613,9E+09,9E+09,9E+09,9E+09,9E+09]], V_rapide, Z_moyen, Tool_Pince1\WObj:=wobj_X62;
    MoveL [[1326.30,577.68,2086.00],[0.308993,-0.00801157,-0.0278477,-0.950623],[0,-1,0,0],[109.267,9E+09,9E+09,9E+09,9E+09,9E+09]],V_rapide,Z_moyen,Tool_Pince1\WObj:=wobj_X62;
    !
    SR_SOUDER lscs2002838300,V_moyen,1,2,Tool_Pince1,wobj_X62;
    SR_SOUDER lspac002872000,V_moyen,1,2,Tool_Pince1,wobj_X62;
    SR_SOUDER lspac002871900,V_moyen,1,1,Tool_Pince1,wobj_X62;
    SR_SOUDER lspac002871800,V_moyen,1,2,Tool_Pince1,wobj_X62;
    SR_SOUDER lspac002871700,V_moyen,1,2,Tool_Pince1,wobj_X62;
    SR_SOUDER lspac002871600,V_moyen,1,2,Tool_Pince1,wobj_X62;
    SR_SOUDER lspac002871500,V_moyen,1,2,Tool_Pince1,wobj_X62;
    SR_SOUDER lspac002871400,V_moyen,1,2,Tool_Pince1,wobj_X62;
    SR_SOUDER lspac002871300,V_moyen,1,1,Tool_Pince1,wobj_X62;
    SR_SOUDER lspac002871200,V_moyen,1,2,Tool_Pince1,wobj_X62;
    SR_SOUDER lspac002871100,V_moyen,1,2,Tool_Pince1,wobj_X62;
    SR_SOUDER lspac002871000,V_moyen,1,2,Tool_Pince1,wobj_X62;
    SR_SOUDER lspac002870900,V_moyen,1,2,Tool_Pince1,wobj_X62;
    ! Abrir Grampos
    !
  ENDPROC

  !-------------
  PROC T_X62K3E23H2_OP()
    VAR bool bStatus;
    Aff_Traj "T_X62K3E23H2_OP";
    AntiReboucle;
    !
    MoveL lscs1002838100,V_rapide,Z_arret,Tool_Pince1\WObj:=wobj_X62;
    !
    MoveL [[1320.90,-551.06,2076.64],[0.529891,0.0162207,0.0240397,-0.84757],[-1,0,0,0],[160,9E+09,9E+09,9E+09,9E+09,9E+09]],V_rapide,Z_Xlarge,Tool_Pince1\WObj:=wobj_X62;
    MoveL [[1444.81,-562.14,2076.59],[0.52988,0.0162209,0.0240409,-0.847577],[0,0,0,0],[160,9E+09,9E+09,9E+09,9E+09,9E+09]],V_rapide,Z_Xlarge,Tool_Pince1\WObj:=wobj_X62;
    !
    SR_SOUDER lscs1004359200, V_moyen, 1, 15, Tool_Pince1, wobj_X62;
    SR_SOUDER lscsd002940301, V_moyen, 1, 15, Tool_Pince1, wobj_X62;
    !
    MoveL [[1657.48,-655.13,2102.77],[0.605718,2.31913E-06,3.73313E-06,-0.79568],[0,-1,0,0],[175.854,9E+09,9E+09,9E+09,9E+09,9E+09]],V_rapide,Z_Xlarge,Tool_Pince1\WObj:=wobj_X62;
    MoveL [[1756.18,-356.78,2097.29],[0.563283,0.00642045,0.0111805,-0.826163],[0,0,0,0],[160,9E+09,9E+09,9E+09,9E+09,9E+09]],V_rapide,Z_Xlarge,Tool_Pince1\WObj:=wobj_X62;
    MoveL [[1570.08,368.66,2084.88],[0.407169,0.0018781,0.00326897,-0.913345],[0,0,0,0],[183.552,9E+09,9E+09,9E+09,9E+09,9E+09]],V_rapide,Z_Xlarge,Tool_Pince1\WObj:=wobj_X62;
    MoveL [[1497.74,665.67,2049.52],[0.339479,5.36477E-06,-3.25454E-06,-0.940614],[0,0,0,0],[182.439,9E+09,9E+09,9E+09,9E+09,9E+09]],V_rapide,Z_arret,Tool_Pince1\WObj:=wobj_X62;
    !
    ! E13:interferencia2 com K5
    ! O12:fora de interferencia1 com K5
    EVENT\E13;
    ORDRE\O12;
    !
    SR_SOUDER lscs2004359300, V_moyen, 1, 15, Tool_Pince1, wobj_X62;
    !
    ! E13:interferencia2 com K5
    ! O12:fora de interferencia1 com K5
    EVENT\E13;
    ORDRE\O12;
    !
    MoveL [[1497.51,666.06,2050],[0.339478,4.49694E-06,1.60091E-05,-0.940614],[0,0,0,0],[173.51,9E+09,9E+09,9E+09,9E+09,9E+09]],V_rapide,Z_Xlarge,Tool_Pince1\WObj:=wobj_X62;
    MoveL [[2241.00,696.13,2009.86],[0.61209,0.00173825,0.00587948,-0.790764],[0,0,0,0],[182.867,9E+09,9E+09,9E+09,9E+09,9E+09]],V_rapide,Z_Xlarge,Tool_Pince1\WObj:=wobj_X62;
    MoveL [[2315.88,926.04,2052.52],[0.583022,0.0035262,-0.00095696,-0.812449],[0,0,0,0],[180.839,9E+09,9E+09,9E+09,9E+09,9E+09]],V_rapide,Z_Xlarge,Tool_Pince1\WObj:=wobj_X62;
    MoveL [[2181.41,1327.16,2032.09],[0.381242,0.000299882,0.000125925,-0.924475],[0,0,1,0],[183.538,9E+09,9E+09,9E+09,9E+09,9E+09]], V_rapide, Z_moyen, Tool_Pince1\WObj:=wobj_X62;
    MoveJ [[1650.02,1566.65,2799.96],[0.370322,0.000249773,0.000216744,-0.928904],[0,0,1,0],[15,9E+09,9E+09,9E+09,9E+09,9E+09]], V_rapide, Z_moyen, Tool_Pince1\WObj:=wobj_X62;
    MoveJ pInicioX62_Pinca1, V_rapide, Z_arret, Tool_Pince1\WObj:=wobj_X62;
    !
  ENDPROC

  !-------------
  PROC T_X62K3CC()
    VAR bool bStatus;
    Aff_Traj "T_X62K3CC";
    AntiReboucle;
    !
    MoveJ pInicioX62_Pinca1, V_rapide, Z_arret, Tool_Pince1\WObj:=wobj_X62;
    MoveL [[536.75,264.72,2747.25],[0.49226,-0.00563274,-0.00397431,-0.870421],[-1,-1,0,0],[41.1525,9E+09,9E+09,9E+09,9E+09,9E+09]],V_rapide,Z_Xlarge,Tool_Pince1\WObj:=wobj_X62;
    MoveL [[593.09,-206.13,2650.54],[0.703477,-0.0059621,-0.00251816,-0.710689],[-1,-1,-1,0],[47.0571,9E+09,9E+09,9E+09,9E+09,9E+09]],V_rapide,Z_Xlarge,Tool_Pince1\WObj:=wobj_X62;
    MoveL [[916.82,1188.70,2645.36],[0.778976,-0.00685561,-0.00263763,-0.627011],[-1,0,-1,0],[47.0568,9E+09,9E+09,9E+09,9E+09,9E+09]],V_rapide,Z_Xlarge,Tool_Pince1\WObj:=wobj_X62;
    MoveL [[922.90,1153.79,1794.34],[0.834184,-0.00707054,-0.00198211,-0.551438],[-1,0,-1,0],[182.764,9E+09,9E+09,9E+09,9E+09,9E+09]],V_rapide,Z_Xlarge,Tool_Pince1\WObj:=wobj_X62;
    MoveL [[1048.21,935.42,1788.67],[0.834182,-0.00705392,-0.00198133,-0.551441],[-1,0,-1,0],[182.764,9E+09,9E+09,9E+09,9E+09,9E+09]], V_moyen, Z_petit, Tool_Pince1\WObj:=wobj_X62;
    MoveL [[1102.24,765.27,1792.23],[0.834181,-0.0070633,-0.00197644,-0.551442],[-1,0,-1,0],[182.764,9E+09,9E+09,9E+09,9E+09,9E+09]], V_moyen, Z_petit, Tool_Pince1\WObj:=wobj_X62;
    MoveL [[1059.94,545.34,1850.51],[0.815681,-0.00569389,-0.0010299,-0.578474],[-1,-1,-1,0],[177.702,9E+09,9E+09,9E+09,9E+09,9E+09]], V_moyen, Z_moyen, Tool_Pince1\WObj:=wobj_X62;
    MoveL [[1059.94,545.34,1850.51],[0.807848,0.07506,0.112769,-0.573613],[-1,-1,-1,0],[177.702,9E+09,9E+09,9E+09,9E+09,9E+09]],V_moyen,Z_moyen,Tool_Pince1\WObj:=wobj_X62;
    MoveL [[1328.58,581.01,1903.25],[0.907214,0.0600704,0.0822127,-0.408161],[-1,-1,-1,0],[172.608,9E+09,9E+09,9E+09,9E+09,9E+09]],V_moyen,Z_moyen,Tool_Pince1\WObj:=wobj_X62;
    MoveL [[1432.18,591.29,1934.15],[0.932451,0.0471665,0.0516043,-0.354468],[-1,-1,-1,0],[171.252,9E+09,9E+09,9E+09,9E+09,9E+09]],V_moyen,Z_moyen,Tool_Pince1\WObj:=wobj_X62;
    !
    MoveL [[1424.74,536.12,1957.61],[0.925341,0.0550874,0.073946,-0.367751],[-1,-1,-1,0],[171.251,9E+09,9E+09,9E+09,9E+09,9E+09]], V_moyen, Z_moyen, Tool_Pince1\WObj:=wobj_X62;
    MoveL [[1438.41,407.58,1970.73],[0.911889,0.0500482,0.066111,-0.401975],[-1,-1,-1,0],[179.15,9E+09,9E+09,9E+09,9E+09,9E+09]],V_moyen,Z_moyen,Tool_Pince1\WObj:=wobj_X62;
    !
    SR_SOUDER lspac002880300, V_moyen, 1, 2, Tool_Pince1, wobj_X62;
    SR_SOUDER lspac002880200, V_moyen, 1, 2, Tool_Pince1, wobj_X62;
    !
    MoveL [[1428.74,204.31,1984.99],[0.877338,0.0294106,0.0218796,-0.478471],[-1,-1,-1,0],[30.0001,9E+09,9E+09,9E+09,9E+09,9E+09]], V_moyen, Z_moyen, Tool_Pince1\WObj:=wobj_X62;
    MoveL [[1431.43,170.40,1982.97],[0.866396,0.029373,0.022812,-0.497971],[-1,-1,-1,0],[30.0015,9E+09,9E+09,9E+09,9E+09,9E+09]], V_moyen, Z_moyen, Tool_Pince1\WObj:=wobj_X62;
    MoveL [[1431.64,170.02,1982.99],[0.855845,0.0288765,0.0234277,-0.515895],[-1,-1,-1,0],[30.0011,9E+09,9E+09,9E+09,9E+09,9E+09]], V_moyen, Z_moyen, Tool_Pince1\WObj:=wobj_X62;
    !
    SR_SOUDER lspac002880100, V_moyen, 1, 2, Tool_Pince1, wobj_X62;
    SR_SOUDER lspac002880000, V_moyen, 1, 2, Tool_Pince1, wobj_X62;
    SR_SOUDER lspac002879900, V_moyen, 1, 2, Tool_Pince1, wobj_X62;
    SR_SOUDER lspac002879800, V_moyen, 1, 2, Tool_Pince1, wobj_X62;
    SR_SOUDER lspac002879700, V_moyen, 1, 2, Tool_Pince1, wobj_X62;
    SR_SOUDER lspac002879600, V_moyen, 1, 2, Tool_Pince1, wobj_X62;
    SR_SOUDER lspac002879500, V_moyen, 1, 2, Tool_Pince1, wobj_X62;
    SR_SOUDER lscs1002847500, V_moyen, 1, 2, Tool_Pince1, wobj_X62;
    SR_SOUDER lscs1002858300, V_moyen, 1, 2, Tool_Pince1, wobj_X62;
    MoveL [[1504.82,-657.46,1962.00],[0.810858,0.0119106,-0.00435938,-0.585106],[-1,0,-1,0],[42.6776,9E+09,9E+09,9E+09,9E+09,9E+09]], V_rapide, Z_moyen, Tool_Pince1\WObj:=wobj_X62;
    MoveL [[1513.37,-694.96,1962.28],[0.804936,0.0124859,-0.0035432,-0.593219],[-1,0,-1,0],[42.6765,9E+09,9E+09,9E+09,9E+09,9E+09]], V_rapide, Z_moyen, Tool_Pince1\WObj:=wobj_X62;
    SR_SOUDER lspac002880400, V_moyen, 1, 2, Tool_Pince1, wobj_X62;
    MoveL [[1492.19,-637.75,1970.56],[0.804936,0.0124997,-0.00352463,-0.59322],[-1,0,-1,0],[42.6761,9E+09,9E+09,9E+09,9E+09,9E+09]], V_rapide, Z_moyen, Tool_Pince1\WObj:=wobj_X62;
    !
    MoveL [[1430.10,-639.34,1890.77],[0.810861,0.0119056,-0.00437854,-0.585102],[-1,0,-1,0],[134.313,9E+09,9E+09,9E+09,9E+09,9E+09]], V_rapide, Z_moyen, Tool_Pince1\WObj:=wobj_X62;
    MoveL [[1326.03,-657.21,1846.57],[0.775528,0.0247824,0.0201514,-0.630504],[-1,-1,-1,0],[175,9E+09,9E+09,9E+09,9E+09,9E+09]],V_rapide,Z_moyen,Tool_Pince1\WObj:=wobj_X62;
    !
    SR_SOUDER lscs1004621800,V_moyen,1,2,Tool_Pince1,wobj_X62;
    SR_SOUDER lscs1002858200,V_moyen,1,2,Tool_Pince1,wobj_X62;
    SR_SOUDER lspac002883400,V_moyen,1,2,Tool_Pince1,wobj_X62;
    SR_SOUDER lspac002883500,V_moyen,1,2,Tool_Pince1,wobj_X62;
    SR_SOUDER lspac002883600,V_moyen,1,2,Tool_Pince1,wobj_X62;
    SR_SOUDER lspac002883700,V_moyen,1,2,Tool_Pince1,wobj_X62;
    !
    MoveL [[1311.70,-133.78,1933.32],[0.824075,0.00662806,0.00455893,-0.566423],[-1,-1,-1,0],[87.807,9E+09,9E+09,9E+09,9E+09,9E+09]], V_rapide, Z_moyen, Tool_Pince1\WObj:=wobj_X62;
    !
    SR_SOUDER lspac002883800,V_moyen,1,2,Tool_Pince1,wobj_X62;
    SR_SOUDER lspac002883900,V_moyen,1,2,Tool_Pince1,wobj_X62;
    !
    MoveL [[1280.53,52.80,1992.27],[0.822187,-0.00265833,-0.00184479,-0.569208],[-1,-1,-1,0],[35.0002,9E+09,9E+09,9E+09,9E+09,9E+09]], V_rapide, Z_moyen, Tool_Pince1\WObj:=wobj_X62;
    MoveL [[1271.72,153.55,1989.81],[0.822186,-0.00264967,-0.00184261,-0.569209],[-1,-1,-1,0],[35.0002,9E+09,9E+09,9E+09,9E+09,9E+09]], V_rapide, Z_moyen, Tool_Pince1\WObj:=wobj_X62;
    !
    SR_SOUDER lspac002884000,V_moyen,1,2,Tool_Pince1,wobj_X62;
    !
    MoveL [[1318.91,169.52,1989.26],[0.834546,0.00309787,0.0296294,-0.550132],[-1,-1,-1,0],[34.9997,9E+09,9E+09,9E+09,9E+09,9E+09]], V_rapide, Z_moyen, Tool_Pince1\WObj:=wobj_X62;
    MoveL [[1323.60,169.93,1986.80],[0.868941,0.00876103,0.0358706,-0.493537],[-1,-1,-1,0],[34.9997,9E+09,9E+09,9E+09,9E+09,9E+09]], V_rapide, Z_moyen, Tool_Pince1\WObj:=wobj_X62;
    !
    SR_SOUDER lspac002884100,V_moyen,1,2,Tool_Pince1,wobj_X62;
    SR_SOUDER lspac002884200,V_moyen,1,2,Tool_Pince1,wobj_X62;
    !
    MoveL [[1313.81,542.00,1974.69],[0.861946,0.0108396,0.0342824,-0.505723],[-1,-1,-1,0],[34.9999,9E+09,9E+09,9E+09,9E+09,9E+09]], V_rapide, Z_moyen, Tool_Pince1\WObj:=wobj_X62;
    !
    SR_SOUDER lspac002884300,V_moyen,1,2,Tool_Pince1,wobj_X62;
    SR_SOUDER lscs2002858000,V_moyen,1,2,Tool_Pince1,wobj_X62;
    SR_SOUDER lscs2004621900,V_moyen,1,2,Tool_Pince1,wobj_X62;
    !
    MoveL [[1110.71,600.71,1937.16],[0.810099,-0.00887349,-0.0195527,-0.5859],[-1,0,-1,0],[62.9354,9E+09,9E+09,9E+09,9E+09,9E+09]], V_moyen, Z_moyen, Tool_Pince1\WObj:=wobj_X62;
    MoveL [[1102.24,765.27,1792.23],[0.834181,-0.0070633,-0.00197644,-0.551442],[-1,0,-1,0],[182.764,9E+09,9E+09,9E+09,9E+09,9E+09]], V_moyen, Z_petit, Tool_Pince1\WObj:=wobj_X62;
    MoveL [[1048.21,935.42,1788.67],[0.834182,-0.00705392,-0.00198133,-0.551441],[-1,0,-1,0],[182.764,9E+09,9E+09,9E+09,9E+09,9E+09]], V_moyen, Z_petit, Tool_Pince1\WObj:=wobj_X62;
    MoveL [[922.90,1153.79,1794.34],[0.834184,-0.00707054,-0.00198211,-0.551438],[-1,0,-1,0],[182.764,9E+09,9E+09,9E+09,9E+09,9E+09]],V_rapide,Z_Xlarge,Tool_Pince1\WObj:=wobj_X62;
    MoveL [[916.82,1188.70,2645.36],[0.778976,-0.00685561,-0.00263763,-0.627011],[-1,0,-1,0],[47.0568,9E+09,9E+09,9E+09,9E+09,9E+09]],V_rapide,Z_Xlarge,Tool_Pince1\WObj:=wobj_X62;
    MoveL [[593.09,-206.13,2650.54],[0.703477,-0.0059621,-0.00251816,-0.710689],[-1,-1,-1,0],[47.0571,9E+09,9E+09,9E+09,9E+09,9E+09]],V_rapide,Z_Xlarge,Tool_Pince1\WObj:=wobj_X62;
    MoveL [[536.75,264.72,2747.25],[0.49226,-0.00563274,-0.00397431,-0.870421],[-1,-1,0,0],[41.1525,9E+09,9E+09,9E+09,9E+09,9E+09]],V_rapide,Z_Xlarge,Tool_Pince1\WObj:=wobj_X62;
    MoveJ pInicioX62_Pinca1, V_rapide, Z_arret, Tool_Pince1\WObj:=wobj_X62;
    !
  ENDPROC
    !-------------
  PROC T_SR1_K0_XDF_L2H1()
     VAR bool bStatus;
     Aff_Traj "T_SR1_K0_XDF_L2H1";
     AntiReboucle;
     !
     MoveJ [[1448.62,1818.65,3375.24],[0.003779,0.999816,-0.01819,-0.004833],[-1,-1,0,0],[60,9E+09,9E+09,9E+09,9E+09,9E+09]],V_rapide,Z_large,Tool_defaut\Wobj:=wobj_XDF;
     !
     MoveJ [[-999.71,1793.55,3017.16],[0.045554,-0.013131,-0.011796,-0.998806],[-1,0,0,0],[180,9E+09,9E+09,9E+09,9E+09,9E+09]],V_rapide,Z_moyen,Tool_Pince1\Wobj:=wobj_XDF;
     MoveJ [[726.99,960.67,2994.34],[0.871059,-0.016963,0.00488,-0.49086],[-1,0,-2,0],[180,9E+09,9E+09,9E+09,9E+09,9E+09]],V_rapide,Z_moyen,Tool_Pince1\Wobj:=wobj_XDF;
     MoveL [[880.82,932,1796.69],[0.789209,0.015943,0.015869,-0.613712],[-1,-1,-1,0],[180,9E+09,9E+09,9E+09,9E+09,9E+09]],V_rapide,Z_moyen,Tool_Pince1\Wobj:=wobj_XDF;
     MoveL [[974.33,50.01,1886.89],[0.758641,0.015158,0.016621,-0.65112],[-1,-1,-1,0],[180,9E+09,9E+09,9E+09,9E+09,9E+09]],V_rapide,Z_arret,Tool_Pince1\Wobj:=wobj_XDF;
     MoveL [[1430.25,-602.16,1915.93],[0.827919,0.024711,0.005044,-0.56028],[-1,0,-1,0],[180,9E+09,9E+09,9E+09,9E+09,9E+09]],V_rapide,Z_arret,Tool_Pince1\Wobj:=wobj_XDF;
     !
     SR_SOUDER SCSDD010167,V_rapide,1,1,Tool_Pince1,wobj_XDF;
     !
     MoveL [[1430.25,-602.16,1915.94],[0.824974,0.024684,0.005173,-0.564607],[-1,0,-1,0],[100,9E+09,9E+09,9E+09,9E+09,9E+09]],V_rapide,Z_arret,Tool_Pince1\Wobj:=wobj_XDF;
     MoveL [[1324.67,-602.73,1925.87],[0.7998,0.016217,0.015589,-0.599845],[-1,-1,-1,0],[100,9E+09,9E+09,9E+09,9E+09,9E+09]],V_rapide,Z_arret,Tool_Pince1\Wobj:=wobj_XDF;
     !
     SR_SOUDER SCSDD010165,V_rapide,1,1,Tool_Pince1,wobj_XDF;
     SR_SOUDER SCSCD010317,V_rapide,1,1,Tool_Pince1,wobj_XDF;
     SR_SOUDER SCSCD010318,V_rapide,1,1,Tool_Pince1,wobj_XDF;
     SR_SOUDER SCSCD010331,V_rapide,1,1,Tool_Pince1,wobj_XDF;
     SR_SOUDER SCSCD010319,V_rapide,1,1,Tool_Pince1,wobj_XDF;
     SR_SOUDER SCSCD010320,V_rapide,1,1,Tool_Pince1,wobj_XDF;
     SR_SOUDER SCSCD010321,V_rapide,1,1,Tool_Pince1,wobj_XDF;
     SR_SOUDER SCSCD010322,V_rapide,1,1,Tool_Pince1,wobj_XDF;
     SR_SOUDER SCSCD010310,V_rapide,1,1,Tool_Pince1,wobj_XDF;
     SR_SOUDER SCSCD010311,V_rapide,1,1,Tool_Pince1,wobj_XDF;
     SR_SOUDER SCSCD010312,V_rapide,1,1,Tool_Pince1,wobj_XDF;
     SR_SOUDER SCSCD010330,V_rapide,1,1,Tool_Pince1,wobj_XDF;
     SR_SOUDER SCSCD010313,V_rapide,1,1,Tool_Pince1,wobj_XDF;
     SR_SOUDER SCSCD010314,V_rapide,1,1,Tool_Pince1,wobj_XDF;
     SR_SOUDER SCSDD010166,V_rapide,1,1,Tool_Pince1,wobj_XDF;
     !
     MoveL [[1204.98,540.24,1880.24],[0.834987,0.009454,-0.025984,-0.549575],[-1,0,-1,0],[180,9E+09,9E+09,9E+09,9E+09,9E+09]],V_rapide,Z_arret,Tool_Pince1\Wobj:=wobj_XDF;
     !
     !ABRIR GRAMPOS
  ENDPROC
     !-------------
  PROC T_SR2_K0_XDF_L2H1()
     MoveL deb_SR2_K0_XD_L2H1,V_rapide,Z_moyen,Tool_Pince1\Wobj:=wobj_XDF;
     !
     MoveL [[982.28,343.73,1873.46],[0.782628,0.093602,-0.106593,-0.60611],[-1,0,-1,0],[180,9E+09,9E+09,9E+09,9E+09,9E+09]],V_rapide,Z_moyen,Tool_Pince1\Wobj:=wobj_XDF;
     MoveL [[580.89,368.81,1804.72],[0.627988,0.198147,-0.244598,-0.711717],[-1,0,-1,0],[180,9E+09,9E+09,9E+09,9E+09,9E+09]],V_rapide,Z_moyen,Tool_Pince1\Wobj:=wobj_XDF;
     !
     SR_SOUDER SCSCD009469,V_rapide,1,1,Tool_Pince1,wobj_XDF;
     SR_SOUDER SCSCD009472,V_rapide,1,1,Tool_Pince1,wobj_XDF;
     !
     MoveL [[628.84,444.27,1754.89],[0.633634,0.214935,-0.229558,-0.706834],[-1,0,-1,0],[180,9E+09,9E+09,9E+09,9E+09,9E+09]],V_rapide,Z_moyen,Tool_Pince1\Wobj:=wobj_XDF;
     MoveL [[870.8,769.44,1774],[0.737524,0.134496,-0.121585,-0.650527],[-1,0,-1,0],[180,9E+09,9E+09,9E+09,9E+09,9E+09]],V_rapide,Z_moyen,Tool_Pince1\Wobj:=wobj_XDF;
     MoveL [[841,1007.58,1772.97],[0.737524,0.134496,-0.121585,-0.650527],[-1,0,-1,0],[180,9E+09,9E+09,9E+09,9E+09,9E+09]],V_rapide,Z_moyen,Tool_Pince1\Wobj:=wobj_XDF;
     MoveJ [[855.55,1072.95,2033.52],[0.782011,0.168528,-0.099154,-0.591799],[-1,0,-1,0],[180,9E+09,9E+09,9E+09,9E+09,9E+09]],V_rapide,Z_moyen,Tool_Pince1\Wobj:=wobj_XDF;
     MoveJ [[571.61,866.61,3000.58],[0.871059,-0.016963,0.00488,-0.49086],[-1,0,-1,0],[180,9E+09,9E+09,9E+09,9E+09,9E+09]],V_rapide,Z_moyen,Tool_Pince1\Wobj:=wobj_XDF;
     MoveJ [[-1098.91,1792.11,3019.69],[0.007414,-0.012671,-0.012289,-0.999817],[-1,0,0,0],[180,9E+09,9E+09,9E+09,9E+09,9E+09]],V_rapide,Z_moyen,Tool_Pince1\Wobj:=wobj_XDF;
     MoveJ p_reb_prg,V_rapide,Z_moyen,Tool_defaut\Wobj:=wobj_XDF;
     !
  ENDPROC
     !-------------
  PROC T_SR1_K0_XDF_L2H2()
     VAR bool bStatus;
     Aff_Traj "T_SR1_K0_XDF_L2H2";
     AntiReboucle;
     !
     MoveJ p_reb_prg,V_rapide,Z_arret,Tool_defaut\Wobj:=wobj0;
     !
     ! E13:interferencia2 com K5
     ! O12:fora de interferencia1 com K5
     ! O14:fora de interferencia3 com K5
     EVENT \E13;
     ORDRE\O12\O14;
     !
     MoveJ [[1715.27,1229.78,2956.83],[0.468809,-0.002395,-0.005648,-0.883278],[0,-1,0,0],[180,9E+09,9E+09,9E+09,9E+09,9E+09]],V_rapide,Z_moyen,Tool_Pince1\Wobj:=wobj_XDF;
     !
     ! E13:interferencia2 com K5
     ! O12:fora de interferencia1 com K5
     ! O14:fora de interferencia3 com K5
     EVENT \E13;
     ORDRE\O12\O14;
     !
     MoveJ [[2279.94,1051.36,2021.06],[0.488012,0.056158,-0.010077,-0.87097],[0,0,0,0],[180,9E+09,9E+09,9E+09,9E+09,9E+09]],V_rapide,Z_moyen,Tool_Pince1\Wobj:=wobj_XDF;
     MoveJ [[1879.7,818.15,2012.33],[0.36029,0.066405,-0.031975,-0.929924],[0,0,0,0],[180,9E+09,9E+09,9E+09,9E+09,9E+09]],V_rapide,Z_moyen,Tool_Pince1\Wobj:=wobj_XDF;
     MoveJ [[1573.63,567.05,2070.5],[0.349111,0.050076,-0.035423,-0.935072],[0,0,0,0],[180,9E+09,9E+09,9E+09,9E+09,9E+09]],V_rapide,Z_moyen,Tool_Pince1\Wobj:=wobj_XDF;
     !
     ! O12:fora de interferencia1 com K5
     ! O13:fora de interferencia2 com K5
     ! O14:fora de interferencia3 com K5
     ORDRE\O12\O13\O14;
     !
     MoveJ [[1416.49,554.78,2100.57],[0.343269,0.041619,-0.037195,-0.937577],[0,0,0,0],[180,9E+09,9E+09,9E+09,9E+09,9E+09]],V_rapide,Z_moyen,Tool_Pince1\Wobj:=wobj_XDF;
     MoveL [[1291.5,556.09,2100.57],[0.302046,0.043202,-0.035344,-0.951658],[0,0,0,0],[180,9E+09,9E+09,9E+09,9E+09,9E+09]],V_rapide,Z_arret,Tool_Pince1\Wobj:=wobj_XDF;
     !
     SR_SOUDER SCS2D035686_L2H2,V_rapide,1,1,Tool_Pince1,wobj_XDF;
     SR_SOUDER SCSCD009431_L2H2,V_rapide,1,1,Tool_Pince1,wobj_XDF;
     SR_SOUDER SCSCD009433_L2H2,V_rapide,1,1,Tool_Pince1,wobj_XDF;
     SR_SOUDER SCSCD009430_L2H2,V_rapide,1,1,Tool_Pince1,wobj_XDF;
     SR_SOUDER SCSCD009432_L2H2,V_rapide,1,1,Tool_Pince1,wobj_XDF;
     SR_SOUDER SCS1D035684_L2H2,V_rapide,1,1,Tool_Pince1,wobj_XDF;
     !
     MoveL [[1301.19,-552.75,2056.09],[0.540273,0.055438,-0.013487,-0.839553],[-1,0,0,0],[180,9E+09,9E+09,9E+09,9E+09,9E+09]],V_rapide,Z_arret,Tool_Pince1\Wobj:=wobj_XDF;
     MoveL [[2235.38,598.90,2176.96],[0.643729,-0.0112334,-0.0186113,-0.764945],[0,-1,0,0],[180,9E+09,9E+09,9E+09,9E+09,9E+09]],V_rapide,Z_moyen,Tool_Pince1\Wobj:=wobj_XDF;
     !
     MoveL [[2445.89,930.94,2158.34],[0.640671,-0.0111625,-0.0186473,-0.767508],[0,-1,0,0],[180.005,9E+09,9E+09,9E+09,9E+09,9E+09]], V_rapide, Z_moyen, Tool_Pince1\WObj:=wobj_XDF;
     MoveJ [[2279.94,1051.36,2021.06],[0.488012,0.056158,-0.010077,-0.87097],[0,0,0,0],[180,9E+09,9E+09,9E+09,9E+09,9E+09]],V_rapide,Z_moyen,Tool_Pince1\Wobj:=wobj_XDF;
     !
     MoveJ [[1715.27,1229.78,2956.83],[0.468809,-0.002395,-0.005648,-0.883278],[0,-1,0,0],[180,9E+09,9E+09,9E+09,9E+09,9E+09]],V_rapide,Z_moyen,Tool_Pince1\Wobj:=wobj_XDF;
     !
     MoveJ p_reb_prg,V_rapide,Z_arret,Tool_defaut\Wobj:=wobj0;
     !ESPERA OPERADOR CARREGAR TETO DIANTEIRO
  ENDPROC
     !-------------
  PROC T_SR2_K0_XDF_L2H2()
     VAR bool bStatus;
     Aff_Traj "T_SR2_K0_XDF_L2H2";
     AntiReboucle;
     !
     MoveJ p_reb_prg,V_rapide,Z_arret,Tool_defaut\Wobj:=wobj0;
     !
     ! E13:interferencia2 com K5
     ! O12:fora de interferencia1 com K5
     ! O14:fora de interferencia3 com K5
     EVENT \E13;
     ORDRE\O12\O14;
     !
     MoveJ [[1715.27,1229.78,2956.83],[0.468809,-0.002395,-0.005648,-0.883278],[0,-1,0,0],[180,9E+09,9E+09,9E+09,9E+09,9E+09]],V_rapide,Z_moyen,Tool_Pince1\Wobj:=wobj_XDF;
     MoveJ [[2279.94,1051.36,2021.06],[0.488012,0.056158,-0.010077,-0.87097],[0,0,0,0],[180,9E+09,9E+09,9E+09,9E+09,9E+09]],V_rapide,Z_moyen,Tool_Pince1\Wobj:=wobj_XDF;
     !
     ! E13:interferencia2 com K5
     ! O12:fora de interferencia1 com K5
     ! O14:fora de interferencia3 com K5
     EVENT \E13;
     ORDRE\O12\O14;
     !
     MoveL [[2259.98,783.90,2107.70],[0.580738,0.026465,-0.0224562,-0.81335],[0,0,0,0],[135.024,9E+09,9E+09,9E+09,9E+09,9E+09]], V_rapide, Z_moyen, Tool_Pince1\WObj:=wobj_XDF;
     MoveJ [[2235.4,598.9,2176.97],[0.682905,-0.012195,-0.018,-0.730184],[0,-1,0,0],[80,9E+09,9E+09,9E+09,9E+09,9E+09]],V_rapide,Z_large,Tool_Pince1\Wobj:=wobj_XDF;
     !
     SR_SOUDER SCS2D011236_L2H2,V_rapide,1,1,Tool_Pince1,wobj_XDF;
     SR_SOUDER SCSCD009371_L2H2,V_rapide,1,1,Tool_Pince1,wobj_XDF;
     !
     MoveJ [[2235.71,596.96,2132.02],[0.682905,-0.012195,-0.018,-0.730184],[0,-1,0,0],[100,9E+09,9E+09,9E+09,9E+09,9E+09]],V_rapide,Z_arret,Tool_Pince1\Wobj:=wobj_XDF;
     MoveJ [[2130.21,599.75,2126.17],[0.682892,-0.012768,-0.018144,-0.730182],[0,-1,0,0],[100,9E+09,9E+09,9E+09,9E+09,9E+09]],V_rapide,Z_arret,Tool_Pince1\Wobj:=wobj_XDF;
     !
     SR_SOUDER SCSCD009369_L2H2,V_rapide,1,1,Tool_Pince1,wobj_XDF;
     SR_SOUDER SCS2D011237_L2H2,V_rapide,1,1,Tool_Pince1,wobj_XDF;
     !
     MoveL [[1291.71,-509.8,2103.8],[0.515047,0.004815,-0.024106,-0.856809],[-1,0,0,0],[100,9E+09,9E+09,9E+09,9E+09,9E+09]],V_rapide,Z_arret,Tool_Pince1\Wobj:=wobj_XDF;
     !
     ! E13:interferencia2 com K5
     ! O12:fora de interferencia1 com K5
     ! O14:fora de interferencia3 com K5
     EVENT \E13;
     ORDRE\O12\O14;
     !
     SR_SOUDER SCSCD009480_L2H2,V_rapide,1,1,Tool_Pince1,wobj_XDF;
     SR_SOUDER SCSCD009487_L2H2,V_rapide,1,1,Tool_Pince1,wobj_XDF;
     SR_SOUDER SCSCD009486_L2H2,V_rapide,1,1,Tool_Pince1,wobj_XDF;
     SR_SOUDER SCSCD009485_L2H2,V_rapide,1,1,Tool_Pince1,wobj_XDF;
     SR_SOUDER SCSCD009482_L2H2,V_rapide,1,1,Tool_Pince1,wobj_XDF;
     SR_SOUDER SCSCD009481_L2H2,V_rapide,1,1,Tool_Pince1,wobj_XDF;
     SR_SOUDER SCSCD009483_L2H2,V_rapide,1,1,Tool_Pince1,wobj_XDF;
     SR_SOUDER SCSCD009484_L2H2,V_rapide,1,1,Tool_Pince1,wobj_XDF;
     SR_SOUDER SCSCD009477_L2H2,V_rapide,1,1,Tool_Pince1,wobj_XDF;
     !
     MoveL [[1258.38,631.48,2142.01],[0.269487,0.0394814,-0.0442899,-0.961175],[0,0,0,0],[20.0012,9E+09,9E+09,9E+09,9E+09,9E+09]],V_rapide,Z_arret,Tool_Pince1\Wobj:=wobj_XDF;
     !
     !COLISAO GRUPO FORA SIMULACAO
     !MoveL [[1284.15,648.14,2131.02],[0.283548,0.055563,-0.039899,-0.956515],[0,0,0,0],[20,9E+09,9E+09,9E+09,9E+09,9E+09]],V_rapide,Z_arret,Tool_Pince1\Wobj:=wobj_XDF;
     !
     !SR_SOUDER SCSCD009478_L2H2,V_rapide,1,1,Tool_Pince1,wobj_XDF;
     !
     !MoveL [[1263.91,631.68,2111.91],[0.273877,0.038442,-0.045202,-0.959933],[0,0,0,0],[100,9E+09,9E+09,9E+09,9E+09,9E+09]],V_rapide,Z_moyen,Tool_Pince1\Wobj:=wobj_XDF;
     !
     MoveL [[1283.98,557.74,2082.83],[0.300198,0.054136,-0.041814,-0.951421],[0,0,0,0],[100,9E+09,9E+09,9E+09,9E+09,9E+09]],V_rapide,Z_moyen,Tool_Pince1\Wobj:=wobj_XDF;
     MoveJ [[1443.51,545.54,2101.1],[0.349606,0.024088,-0.036021,-0.935894],[0,0,0,0],[100,9E+09,9E+09,9E+09,9E+09,9E+09]],V_rapide,Z_moyen,Tool_Pince1\Wobj:=wobj_XDF;
     MoveL [[1452.74,684.01,2135.53],[0.309066,0.003801,-0.035714,-0.950362],[0,0,0,0],[100,9E+09,9E+09,9E+09,9E+09,9E+09]],V_rapide,Z_arret,Tool_Pince1\Wobj:=wobj_XDF;
     !
     SR_SOUDER SCS2D010234_L2H2,V_rapide,1,1,Tool_Pince1,wobj_XDF;
     !
     MoveJ [[1452.74,684.01,2135.53],[0.299968,0.023449,-0.036439,-0.952965],[0,0,0,0],[20,9E+09,9E+09,9E+09,9E+09,9E+09]], V_rapide, Z_arret, Tool_Pince1\WObj:=wobj_XDF;
     !
     SR_SOUDER SCSCD009429_L2H2,V_rapide,1,1,Tool_Pince1,wobj_XDF;
     SR_SOUDER SCSCD009427_L2H2,V_rapide,1,1,Tool_Pince1,wobj_XDF;
     SR_SOUDER SCSCD009434_L2H2,V_rapide,1,1,Tool_Pince1,wobj_XDF;
     SR_SOUDER SCSCD009428_L2H2,V_rapide,1,1,Tool_Pince1,wobj_XDF;
     SR_SOUDER SCSCD009422_L2H2,V_rapide,1,1,Tool_Pince1,wobj_XDF;
     SR_SOUDER SCSCD009421_L2H2,V_rapide,1,1,Tool_Pince1,wobj_XDF;
     SR_SOUDER SCSCD009426_L2H2,V_rapide,1,1,Tool_Pince1,wobj_XDF;
     SR_SOUDER SCS1D035683_L2H2_,V_rapide,1,1,Tool_Pince1,wobj_XDF;
     !
     MoveJ [[1459.99,-565.59,2120.92],[0.501271,0.042073,-0.016812,-0.864103],[0,0,0,0],[50,9E+09,9E+09,9E+09,9E+09,9E+09]],V_rapide,Z_large,Tool_Pince1\Wobj:=wobj_XDF;
     !
     SR_SOUDER SCS1D009539_L2H2,V_rapide,1,1,Tool_Pince1,wobj_XDF;
     SR_SOUDER SCS1D009551_L2H2,V_rapide,1,1,Tool_Pince1,wobj_XDF;
     SR_SOUDER SCS1D009540_L2H2,V_rapide,1,1,Tool_Pince1,wobj_XDF;
     SR_SOUDER SCS1D009541_L2H2,V_rapide,1,1,Tool_Pince1,wobj_XDF;
     SR_SOUDER SCS1D009542_L2H2,V_rapide,1,1,Tool_Pince1,wobj_XDF;
     !
     MoveL [[1814.25,-588.61,2129.34],[0.570362,0.021113,0.015787,-0.82097],[0,0,0,0],[50,9E+09,9E+09,9E+09,9E+09,9E+09]],V_rapide,Z_large,Tool_Pince1\Wobj:=wobj_XDF;
     !
     SR_SOUDER SCSCD009372_L2H2,V_rapide,1,1,Tool_Pince1,wobj_XDF;
     SR_SOUDER SCSCD009361_L2H2,V_rapide,1,1,Tool_Pince1,wobj_XDF;
     SR_SOUDER SCSCD009374_L2H2,V_rapide,1,1,Tool_Pince1,wobj_XDF;
     SR_SOUDER SCSCD009373_L2H2,V_rapide,1,1,Tool_Pince1,wobj_XDF;
     !
     MoveJ [[2136.26,-14.44,2145.55],[0.587632,0.004571,-0.002417,-0.809111],[0,0,0,0],[80,9E+09,9E+09,9E+09,9E+09,9E+09]],V_rapide,Z_arret,Tool_Pince1\Wobj:=wobj_XDF;
     MoveJ [[2231.24,0.05,2146.4],[0.643317,0.003297,-0.001961,-0.76559],[0,0,0,0],[80,9E+09,9E+09,9E+09,9E+09,9E+09]],V_rapide,Z_arret,Tool_Pince1\Wobj:=wobj_XDF;
     !
     SR_SOUDER SCSCD009363_L2H2,V_rapide,1,1,Tool_Pince1,wobj_XDF;
     SR_SOUDER SCSCD009362_L2H2,V_rapide,1,1,Tool_Pince1,wobj_XDF;
     SR_SOUDER SCSCD009370_L2H2,V_rapide,1,1,Tool_Pince1,wobj_XDF;
     SR_SOUDER SCSCD009360_L2H2,V_rapide,1,1,Tool_Pince1,wobj_XDF;
     SR_SOUDER SCSCD009358_L2H2,V_rapide,1,1,Tool_Pince1,wobj_XDF;
     SR_SOUDER SCS1D011234_L2H2,V_rapide,1,1,Tool_Pince1,wobj_XDF;
     !
     MoveJ [[2235.4,-598.9,2131.97],[0.706888,0.017586,0.012787,-0.706991],[0,0,0,0],[100,9E+09,9E+09,9E+09,9E+09,9E+09]],V_rapide,Z_arret,Tool_Pince1\Wobj:=wobj_XDF;
     MoveJ [[2183.8,-697.21,2118.51],[0.706829,0.020657,0.014551,-0.706933],[0,0,0,0],[100,9E+09,9E+09,9E+09,9E+09,9E+09]],V_rapide,Z_arret,Tool_Pince1\Wobj:=wobj_XDF;
     !
     SR_SOUDER SCS1D009546_L2H2,V_rapide,1,1,Tool_Pince1,wobj_XDF;
     !
     MoveL [[2183.8,-697.21,2118.51],[0.706829,0.020657,0.014551,-0.706933],[0,0,0,0],[100,9E+09,9E+09,9E+09,9E+09,9E+09]],V_rapide,Z_large,Tool_Pince1\Wobj:=wobj_XDF;
     !
     SR_SOUDER SCS1D009547_L2H2,V_rapide,1,1,Tool_Pince1,wobj_XDF;
     SR_SOUDER SCS1D009548_L2H2,V_rapide,1,1,Tool_Pince1,wobj_XDF;
     SR_SOUDER SCS1D009549_L2H2,V_rapide,1,1,Tool_Pince1,wobj_XDF;
     SR_SOUDER SCS1D009553_L2H2,V_rapide,1,1,Tool_Pince1,wobj_XDF;
     SR_SOUDER SCS1D009552_L2H2,V_rapide,1,1,Tool_Pince1,wobj_XDF;
     !
     MoveJ [[2787.74,-698.4,2152.09],[0.725092,0.02021,0.017347,-0.688137],[0,0,0,0],[180,9E+09,9E+09,9E+09,9E+09,9E+09]],V_rapide,Z_large,Tool_Pince1\Wobj:=wobj_XDF;
     MoveL [[3009.34,-696.44,2123.21],[0.793095,0.02015,0.014943,-0.608581],[0,0,0,0],[180,9E+09,9E+09,9E+09,9E+09,9E+09]],V_rapide,Z_arret,Tool_Pince1\Wobj:=wobj_XDF;
     !
     SR_SOUDER SCS1D009927_L2H2,V_rapide,1,1,Tool_Pince1,wobj_XDF;
     !
     MoveJ [[3009.34,-696.44,2123.21],[0.793095,0.02015,0.014943,-0.608581],[0,0,0,0],[180,9E+09,9E+09,9E+09,9E+09,9E+09]],V_rapide,Z_arret,Tool_Pince1\Wobj:=wobj_XDF;
     MoveL [[2957.25,-621.56,2135.44],[0.818762,0.018267,0.013513,-0.573683],[0,0,0,0],[150,9E+09,9E+09,9E+09,9E+09,9E+09]],V_rapide,Z_arret,Tool_Pince1\Wobj:=wobj_XDF;
     !
     SR_SOUDER SCSCD009418_L2H2,V_rapide,1,1,Tool_Pince1,wobj_XDF;
     SR_SOUDER SCSCD009400_L2H2,V_rapide,1,1,Tool_Pince1,wobj_XDF;
     SR_SOUDER SCSCD009398_L2H2,V_rapide,1,1,Tool_Pince1,wobj_XDF;
     SR_SOUDER SCSCD009408_L2H2,V_rapide,1,1,Tool_Pince1,wobj_XDF;
     SR_SOUDER SCSCD009416_L2H2,V_rapide,1,1,Tool_Pince1,wobj_XDF;
     SR_SOUDER SCSCD009406_L2H2,V_rapide,1,1,Tool_Pince1,wobj_XDF;
     SR_SOUDER SCSCD009414_L2H2,V_rapide,1,1,Tool_Pince1,wobj_XDF;
     SR_SOUDER SCSCD009404_L2H2,V_rapide,1,1,Tool_Pince1,wobj_XDF;
     SR_SOUDER SCSCD009412_L2H2,V_rapide,1,1,Tool_Pince1,wobj_XDF;
     !
     !PEDIDO DE INTERLOCK 1
     !
     ! E12:interferencia1 com K5
     ! O13:fora de interferencia2 com K5
     ! O14:fora de interferencia3 com K5
     EVENT \E12;
     ORDRE\O13\O14;
     !
     SR_SOUDER SCSCD009410_L2H2,V_rapide,1,1,Tool_Pince1,wobj_XDF;
     !
     ! E12:interferencia1 com K5
     ! O13:fora de interferencia2 com K5
     ! O14:fora de interferencia3 com K5
     EVENT \E12;
     ORDRE\O13\O14;
     !
     SR_SOUDER SCSCD009396_L2H2,V_rapide,1,1,Tool_Pince1,wobj_XDF;
     SR_SOUDER SCSCD009402_L2H2,V_rapide,1,1,Tool_Pince1,wobj_XDF;
     SR_SOUDER SCSCD009420_L2H2,V_rapide,1,1,Tool_Pince1,wobj_XDF;
     !
     MoveL [[2957.24,621.56,2135.44],[0.942107,-0.021601,-0.007036,-0.334541],[0,-1,-1,0],[100,9E+09,9E+09,9E+09,9E+09,9E+09]],V_rapide,Z_arret,Tool_Pince1\Wobj:=wobj_XDF;
     MoveL [[3062.43,573.54,2137.6],[0.927159,-0.018991,-0.008065,-0.374099],[0,-1,-1,0],[100,9E+09,9E+09,9E+09,9E+09,9E+09]],V_rapide,Z_arret,Tool_Pince1\Wobj:=wobj_XDF;
     !
     SR_SOUDER SCSCD009382_L2H2,V_rapide,1,1,Tool_Pince1,wobj_XDF;
     SR_SOUDER SCSCD009384_L2H2,V_rapide,1,1,Tool_Pince1,wobj_XDF;
     SR_SOUDER SCSCD009394_L2H2,V_rapide,1,1,Tool_Pince1,wobj_XDF;
     SR_SOUDER SCSCD009378_L2H2,V_rapide,1,1,Tool_Pince1,wobj_XDF;
     !
     !FORA DE INTERFERENCIA 1
     !
     ! O12:fora de interferencia1 com K5
     ! O13:fora de interferencia2 com K5
     ! O14:fora de interferencia3 com K5
     ORDRE\O12\O13\O14;
     !3
     SR_SOUDER SCSCD009386_L2H2,V_rapide,1,1,Tool_Pince1,wobj_XDF;
     SR_SOUDER SCSCD009380_L2H2,V_rapide,1,1,Tool_Pince1,wobj_XDF;
     SR_SOUDER SCSCD009392_L2H2,V_rapide,1,1,Tool_Pince1,wobj_XDF;
     SR_SOUDER SCSCD009388_L2H2,V_rapide,1,1,Tool_Pince1,wobj_XDF;
     SR_SOUDER SCSCD009390_L2H2,V_rapide,1,1,Tool_Pince1,wobj_XDF;
     SR_SOUDER SCSGD010159_L2H2,V_rapide,1,1,Tool_Pince1,wobj_XDF;
     SR_SOUDER SCS1D010180_L2H2,V_rapide,1,1,Tool_Pince1,wobj_XDF;
     !
     MoveL [[3065.53,-600.23,2181.55],[0.819925,0.019069,0.012864,-0.572008],[0,0,0,0],[80,9E+09,9E+09,9E+09,9E+09,9E+09]],V_rapide,Z_arret,Tool_Pince1\Wobj:=wobj_XDF;
     !
     !ABRIR GRAMPOS
  ENDPROC
     !-------------
  PROC T_SR3_K0_XDF_L2H2()
     MoveJ [[3065.53,-600.23,2181.55],[0.819925,0.019069,0.012864,-0.572008],[0,0,0,0],[100,9E+09,9E+09,9E+09,9E+09,9E+09]],V_rapide,Z_arret,Tool_Pince1\Wobj:=wobj_XDF;
     !
     ! O12:fora de interferencia1 com K5
     ! O13:fora de interferencia2 com K5
     ! O14:fora de interferencia3 com K5
     ORDRE\O12\O13\O14;
     !
     !ABRIR GRAMPOS
     MoveJ [[2907.48,-698.92,2121.88],[0.793075,0.0209433,0.014997,-0.608579],[0,0,0,0],[130.809,9E+09,9E+09,9E+09,9E+09,9E+09]],V_rapide,Z_arret,Tool_Pince1\Wobj:=wobj_XDF;
     !
     SR_SOUDER SCS1D009550_L2H2,V_rapide,1,1,Tool_Pince1,wobj_XDF;
     !
     MoveL [[2136.63,-572.83,2133.78],[0.706939,0.016518,0.009734,-0.707014],[0,0,0,0],[100,9E+09,9E+09,9E+09,9E+09,9E+09]],V_rapide,Z_arret,Tool_Pince1\Wobj:=wobj_XDF;
     !
     SR_SOUDER SCSCD009359_L2H2,V_rapide,1,1,Tool_Pince1,wobj_XDF;
     SR_SOUDER SCS1D011235_L2H2,V_rapide,1,1,Tool_Pince1,wobj_XDF;
     SR_SOUDER SCS1D009545_L2H2,V_rapide,1,1,Tool_Pince1,wobj_XDF;
     SR_SOUDER SCS1D009544_L2H2,V_rapide,1,1,Tool_Pince1,wobj_XDF;
     SR_SOUDER SCS1D009543_L2H2,V_rapide,1,1,Tool_Pince1,wobj_XDF;
     !
     MoveL [[2057.6,-380.04,2128.58],[0.633068,0.021321,0.014091,-0.773675],[0,0,0,0],[180,9E+09,9E+09,9E+09,9E+09,9E+09]],V_rapide,Z_arret,Tool_Pince1\Wobj:=wobj_XDF;
     !
     ! E13:interferencia2 com K5
     ! O12:fora de interferencia1 com K5
     ! O14:fora de interferencia3 com K5
     EVENT \E13;
     ORDRE\O12\O14;
     !
     MoveL [[2276.28,883.45,2014.74],[0.519239,0.019153,0.016921,-0.854247],[0,0,0,0],[180,9E+09,9E+09,9E+09,9E+09,9E+09]],V_rapide,Z_arret,Tool_Pince1\Wobj:=wobj_XDF;
     MoveJ [[941.05,1190.48,1286.22],[0.013707,0.271873,0.961968,0.022674],[0,-1,0,0],[180,9E+09,9E+09,9E+09,9E+09,9E+09]],V_rapide,Z_arret,Tool_defaut\Wobj:=wobj0;
     MoveJ [[1921.97,1262.65,2963.64],[0.52407,0.000933911,-0.00195563,-0.851673],[0,-1,0,0],[170.001,9E+09,9E+09,9E+09,9E+09,9E+09]], V_rapide, Z_arret, Tool_Pince1\WObj:=wobj_XDF;
     !
     MoveJ [[434.45,1757.37,2971.08],[0.024116,-0.00434763,-0.000447855,-0.9997],[-1,-1,0,0],[59.9983,9E+09,9E+09,9E+09,9E+09,9E+09]],V_rapide,Z_arret,Tool_Pince1\Wobj:=wobj_XDF;
     !
     ! O12:fora de interferencia1 com K5
     ! O13:fora de interferencia2 com K5
     ! O14:fora de interferencia3 com K5
     ORDRE\O12\O13\O14;
     !
  ENDPROC

!************************** Trajectoires pour changeur d'outils *******************************

  PROC T_RODCYCLE_P1()
    Aff_Traj "T_RODCYCLE_P1";
    AntiReboucle;
    !
    ! Traj rodage Séquenceur 1 pince 1
    MoveJ p_repli, V_moyen, Z_arret, Tool_defaut;
    MoveL [[331.05,-2668.97,-882.88],[0.675747,-0.00563673,0.0008286,-0.737112],[-1,-1,0,0],[137.124,9E+09,9E+09,9E+09,9E+09,9E+09]], V_moyen, Z_moyen, Tool_Pince1;
    MoveL [[329.67,-2817.33,-882.92],[0.675727,-0.00563172,0.000837921,-0.73713],[-1,-1,0,0],[137.124,9E+09,9E+09,9E+09,9E+09,9E+09]], V_moyen, Z_moyen, Tool_Pince1;
    MoveL pFresaPinca1, V_moyen, Z_arret, Tool_Pince1;
    !
    SR_RODER 1,1;
    !
    MoveL [[329.67,-2817.33,-882.92],[0.675727,-0.00563172,0.000837921,-0.73713],[-1,-1,0,0],[137.124,9E+09,9E+09,9E+09,9E+09,9E+09]], V_moyen, Z_moyen, Tool_Pince1;
    MoveL [[331.05,-2668.97,-882.88],[0.675747,-0.00563673,0.0008286,-0.737112],[-1,-1,0,0],[137.124,9E+09,9E+09,9E+09,9E+09,9E+09]], V_moyen, Z_moyen, Tool_Pince1;
    MoveJ p_repli, V_moyen, Z_arret, Tool_defaut;
    !
    SR_INIT_PINCE 1;
    SR_SOUDER p_repli, V_moyen, 1, 255, Tool_defaut, wobj0;
    !
  ENDPROC

  !------------
  !Enlever les commentaires pour l'option Changeur Outil
!  PROC T_ROD_1()
!    SR_SERVICE 1\AppelTraj:="T_ROD_P1";
!    SR_SERVICE 2\AppelTraj:="T_ROD_P2";
!    SR_SERVICE 3\AppelTraj:="T_ROD_P3";
!    SR_SERVICE 4\AppelTraj:="T_ROD_P4";
!  ENDPROC

  PROC T_ROD_P1()
    Aff_Traj "T_ROD_P1";
    AntiReboucle;
    ! Traj rodage Séquenceur 1 pince 1
    MoveJ p_reb_prg,V_moyen,Z_arret,Tool_defaut;
    SR_RODER 1,141;
    ! trajectoire dégagement
    SR_INIT_PINCE 1;
    SR_SOUDER p_reb_prg, V_moyen, 1,151, Tool_defaut, wobj0;
  ENDPROC

  PROC T_ROD_P2()
    Aff_Traj "T_ROD_P2";
    AntiReboucle;
    ! Traj rodage Séquenceur 1 pince 2
    MoveJ p_reb_prg,V_moyen,Z_arret,Tool_defaut;
    SR_RODER 2,142;
    ! trajectoire dégagement
    SR_INIT_PINCE 2;
    SR_SOUDER p_reb_prg, V_moyen, 2,152, Tool_defaut, wobj0;
  ENDPROC

  PROC T_ROD_P3()
    Aff_Traj "T_ROD_P3";
    AntiReboucle;
    ! Traj rodage Séquenceur 1 pince 3
    MoveJ p_reb_prg,V_moyen,Z_arret,Tool_defaut;
    SR_RODER 3,143;
    ! trajectoire dégagement
    SR_INIT_PINCE 3;
    SR_SOUDER p_reb_prg, V_moyen, 3,153, Tool_defaut, wobj0;
  ENDPROC

  PROC T_ROD_P4()
    Aff_Traj "T_ROD_P4";
    AntiReboucle;
    ! Traj rodage Séquenceur 1 pince 4
    MoveJ p_reb_prg,V_moyen,Z_arret,Tool_defaut;
    SR_RODER 4,144;
    ! trajectoire dégagement
    SR_INIT_PINCE 4;
    SR_SOUDER p_reb_prg, V_moyen, 4,154, Tool_defaut, wobj0;
  ENDPROC

  !------------
  !Enlever les commentaires pour l'option Changeur Outil
!  PROC T_Chelm1()
!    SR_SERVICE 1\AppelTraj:="T_CHELM_P1";
!    SR_SERVICE 2\AppelTraj:="T_CHELM_P2";
!    SR_SERVICE 3\AppelTraj:="T_CHELM_P3";
!    SR_SERVICE 4\AppelTraj:="T_CHELM_P4";
!  ENDPROC

  !------------
  PROC T_CHELM_P1()
    Aff_Traj "T_CHELM_P1";
    AntiReboucle;
    ! Traj chgt manu séquenceur 1 Pince 1
    MoveJ p_reb_prg,V_moyen,Z_arret,Tool_defaut;
    SR_CEAU 1;
    ! Trajectoire approche
    SR_CHELMAN 1;
    SR_CEAU 0;
    ! trajectoire dégagement
    SR_INIT_PINCE 1;
    SR_SOUDER p_reb_prg,V_moyen,1,151,Tool_defaut,wobj0;
    AutoriseTraj;
    T_Usinage_P1;
  ENDPROC

  !------------
  PROC T_CHELM_P2()
    Aff_Traj "T_CHELM_P2";
    AntiReboucle;
    ! Traj chgt manu séquenceur 1 Pince 2
    MoveJ p_reb_prg,V_moyen,Z_arret,Tool_defaut;
    SR_CEAU 1;
    ! Trajectoire approche
    SR_CHELMAN 2;
    SR_CEAU 0;
    ! trajectoire dégagement
    SR_INIT_PINCE 2;
    SR_SOUDER p_reb_prg,V_moyen,2,152,Tool_defaut,wobj0;
    AutoriseTraj;
    T_Usinage_P2;
  ENDPROC

  !------------
  PROC T_CHELM_P3()
    Aff_Traj "T_CHELM_P3";
    AntiReboucle;
    ! Traj chgt manu séquenceur 1 Pince 3
    MoveJ p_reb_prg,V_moyen,Z_arret,Tool_defaut;
    SR_CEAU 1;
    ! Trajectoire approche
    SR_CHELMAN 3;
    SR_CEAU 0;
    ! trajectoire dégagement
    SR_INIT_PINCE 3;
    SR_SOUDER p_reb_prg,V_moyen,3,153,Tool_defaut,wobj0;
    AutoriseTraj;
    T_Usinage_P3;
  ENDPROC

  !------------
  PROC T_CHELM_P4()
    Aff_Traj "T_CHELM_P4";
    AntiReboucle;
    ! Traj chgt manu séquenceur 1 Pince 4
    MoveJ p_reb_prg,V_moyen,Z_arret,Tool_defaut;
    SR_CEAU 1;
    ! Trajectoire approche
    SR_CHELMAN 4;
    SR_CEAU 0;
    ! trajectoire dégagement
    SR_INIT_PINCE 4;
    SR_SOUDER p_reb_prg,V_moyen,4,154,Tool_defaut,wobj0;
    AutoriseTraj;
    T_Usinage_P4;
  ENDPROC

  !------------
  PROC T_Usinage_P1()
    Aff_Traj "T_Usinage_P1";
    AntiReboucle;
    ! Traj usinage séquenceur 1 Pince 1
    MoveJ p_reb_prg,V_moyen,Z_arret,Tool_defaut;
    ! Trajectoire approche
    SR_RODER 1,131;
    ! trajectoire dégagement
    SR_INIT_PINCE 1;
    SR_SOUDER p_reb_prg,V_moyen,1,151,Tool_defaut,wobj0;
  ENDPROC

  !------------
  PROC T_Usinage_P2()
    Aff_Traj "T_Usinage_P2";
    AntiReboucle;
    ! Traj usinage séquenceur 1 Pince 2
    MoveJ p_reb_prg,V_moyen,Z_arret,Tool_defaut;
    ! Trajectoire approche
    SR_RODER 2,132;
    ! trajectoire dégagement
    SR_INIT_PINCE 2;
    SR_SOUDER p_reb_prg,V_moyen,2,152,Tool_defaut,wobj0;
  ENDPROC

  !------------
  PROC T_Usinage_P3()
    Aff_Traj "T_Usinage_P3";
    AntiReboucle;
    ! Traj usinage séquenceur 1 Pince 3
    MoveJ p_reb_prg,V_moyen,Z_arret,Tool_defaut;
    ! Trajectoire approche
    SR_RODER 3,133;
    ! trajectoire dégagement
    SR_INIT_PINCE 3;
    SR_SOUDER p_reb_prg,V_moyen,3,153,Tool_defaut,wobj0;
  ENDPROC

  !------------
  PROC T_Usinage_P4()
    Aff_Traj "T_Usinage_P4";
    AntiReboucle;
    ! Traj usinage séquenceur 1 Pince 4
    MoveJ p_reb_prg,V_moyen,Z_arret,Tool_defaut;
    ! Trajectoire approche
    SR_RODER 4,134;
    ! trajectoire dégagement
    SR_INIT_PINCE 4;
    SR_SOUDER p_reb_prg,V_moyen,4,154,Tool_defaut,wobj0;
  ENDPROC

  !------------
  PROC T_SEGURANCATRASEIRA()
    toolAtual := CTool();
    wobjAtual := CWObj();
    !
    MoveJ CRobT(), V_moyen, Z_arret, toolAtual\WObj:=wobjAtual;
    ! O9:segurança traseira com K1
    ! O12:fora de interferencia1 com K5
    ! O13:fora de interferencia2 com K5
    ORDRE\O9\O12\O13;
    !
  ENDPROC

  !------------
  PROC T_AUTORIZA_RECUO()
    toolAtual := CTool();
    wobjAtual := CWObj();
    !
    MoveJ CRobT(),V_moyen,Z_arret,toolAtual\WObj:=wobjAtual;
    ! E9:autorização de recuo
    ! O12:fora de interferencia1 com K5
    ! O13:fora de interferencia2 com K5
    EVENT\E9;
    ORDRE\O12\O13;
    !
  ENDPROC

ENDMODULE
